LIN {X 0,Y 429.62,Z 995.465,A -85,B 0,C 180,E1 8895.717,E2 8895.717} C_VEL
LIN {X 0,Y 428.835,Z 1009.272,A -85,B 0,C 180,E1 8900.698,E2 8900.698} C_VEL
LIN {X 0,Y 428.636,Z 1016.168,A -85,B 0,C 180,E1 8904.933,E2 8904.933} C_VEL
LIN {X 0,Y 428.616,Z 1019.114,A -85,B 0,C 180,E1 8910,E2 8910} C_VEL
LIN {X 0,Y 428.715,Z 1016.175,A -85,B 0,C 180,E1 8915.065,E2 8915.065} C_VEL
LIN {X 0,Y 428.851,Z 1009.233,A -85,B 0,C 180,E1 8919.317,E2 8919.317} C_VEL
LIN {X 0,Y 429.678,Z 995.468,A -85,B 0,C 180,E1 8924.28,E2 8924.28} C_VEL
LIN {X 0,Y 431.433,Z 976.764,A -85,B 0,C 180,E1 8928.853,E2 8928.853} C_VEL
LIN {X 0,Y 434.387,Z 952.802,A -85,B 0,C 180,E1 8933.087,E2 8933.087} C_VEL
LIN {X 0,Y 438.277,Z 923.802,A -85,B 0,C 180,E1 8936.824,E2 8936.824} C_VEL
LIN {X 0,Y 442.644,Z 891.156,A -85,B 0,C 180,E1 8939.875,E2 8939.875} C_VEL
LIN {X 0,Y 446.524,Z 856.568,A -85,B 0,C 180,E1 8942.13,E2 8942.13} C_VEL
LIN {X 0,Y 449.583,Z 820.465,A -85,B 0,C 180,E1 8943.637,E2 8943.637} C_VEL
LIN {X 0,Y 450.41,Z 794.271,A -85,B 0,C 180,E1 8944.326,E2 8944.326} C_VEL
LIN {X 0,Y 439.203,Z 761.451,A -85,B 0,C 180,E1 8945.976,E2 8945.976} C_VEL
LIN {X 0,Y 430.955,Z 742.619,A -85,B 0,C 180,E1 8947.153,E2 8947.153} C_VEL
LIN {X 0,Y 427.18,Z 733.66,A -85,B 0,C 180,E1 8947.767,E2 8947.767} C_VEL
LIN {X 0,Y 427.055,Z 733.66,A -85,B 0,C 180,E1 8954.849,E2 8954.849} C_VEL
LIN {X 0,Y 427.009,Z 733.66,A -85,B 0,C 180,E1 8961.267,E2 8961.267} C_VEL
LIN {X 0,Y 427.177,Z 733.66,A -85,B 0,C 180,E1 8968.283,E2 8968.283} C_VEL
LIN {X 0,Y 427.333,Z 734.394,A -85,B 0,C 180,E1 8973.698,E2 8973.698} C_VEL
LIN {X 0,Y 436.898,Z 759.131,A -85,B 0,C 180,E1 8975.578,E2 8975.578} C_VEL
LIN {X 0,Y 439.517,Z 771.894,A -85,B 0,C 180,E1 8976.207,E2 8976.207} C_VEL
LIN {X 0,Y 438.674,Z 800.731,A -85,B 0,C 180,E1 8977.463,E2 8977.463} C_VEL
LIN {X 0,Y 437.062,Z 826.317,A -85,B 0,C 180,E1 8979.38,E2 8979.38} C_VEL
LIN {X 0,Y 435.066,Z 849.12,A -85,B 0,C 180,E1 8982.015,E2 8982.015} C_VEL
LIN {X 0,Y 433.123,Z 867.039,A -85,B 0,C 180,E1 8985.093,E2 8985.093} C_VEL
LIN {X 0,Y 431.622,Z 879.714,A -85,B 0,C 180,E1 8988.42,E2 8988.42} C_VEL
LIN {X 0,Y 430.66,Z 887.62,A -85,B 0,C 180,E1 8991.921,E2 8991.921} C_VEL
LIN {X 0,Y 430.105,Z 890.96,A -85,B 0,C 180,E1 8995.967,E2 8995.967} C_VEL
LIN {X 0,Y 430.036,Z 888.324,A -85,B 0,C 180,E1 9000.005,E2 9000.005} C_VEL
LIN {X 0,Y 430.501,Z 879.672,A -85,B 0,C 180,E1 9004.038,E2 9004.038} C_VEL
LIN {X 0,Y 431.437,Z 865.002,A -85,B 0,C 180,E1 9007.82,E2 9007.82} C_VEL
LIN {X 0,Y 432.768,Z 846,A -85,B 0,C 180,E1 9011.013,E2 9011.013} C_VEL
LIN {X 0,Y 434.452,Z 821.904,A -85,B 0,C 180,E1 9013.738,E2 9013.738} C_VEL
LIN {X 0,Y 436.003,Z 794.969,A -85,B 0,C 180,E1 9015.745,E2 9015.745} C_VEL
LIN {X 0,Y 436.384,Z 764.977,A -85,B 0,C 180,E1 9017.084,E2 9017.084} C_VEL
LIN {X 0,Y 427.56,Z 733.66,A -85,B 0,C 180,E1 9018.342,E2 9018.342} C_VEL
LIN {X 0,Y 427.307,Z 733.66,A -85,B 0,C 180,E1 9025.167,E2 9025.167} C_VEL
LIN {X 0,Y 427.11,Z 733.66,A -85,B 0,C 180,E1 9032.127,E2 9032.127} C_VEL
LIN {X 0,Y 426.99,Z 733.66,A -85,B 0,C 180,E1 9038.73,E2 9038.73} C_VEL
LIN {X 0,Y 427.072,Z 733.66,A -85,B 0,C 180,E1 9045.161,E2 9045.161} C_VEL
LIN {X 0,Y 427.062,Z 733.66,A -85,B 0,C 180,E1 9051.262,E2 9051.262} C_VEL
LIN {X 0,Y 427.143,Z 733.808,A -85,B 0,C 180,E1 9052.71,E2 9052.71} C_VEL
LIN {X 0,Y 447.309,Z 778.034,A -85,B 0,C 180,E1 9055.746,E2 9055.746} C_VEL
LIN {X 0,Y 450.534,Z 788.772,A -85,B 0,C 180,E1 9056.452,E2 9056.452} C_VEL
LIN {X 0,Y 447.329,Z 824.927,A -85,B 0,C 180,E1 9058.189,E2 9058.189} C_VEL
LIN {X 0,Y 443.379,Z 857.575,A -85,B 0,C 180,E1 9060.541,E2 9060.541} C_VEL
LIN {X 0,Y 438.938,Z 889.11,A -85,B 0,C 180,E1 9063.751,E2 9063.751} C_VEL
LIN {X 0,Y 434.909,Z 915.634,A -85,B 0,C 180,E1 9067.484,E2 9067.484} C_VEL
LIN {X 0,Y 431.753,Z 938.347,A -85,B 0,C 180,E1 9071.867,E2 9071.867} C_VEL
LIN {X 0,Y 429.91,Z 954.579,A -85,B 0,C 180,E1 9076.248,E2 9076.248} C_VEL
LIN {X 0,Y 428.868,Z 966.988,A -85,B 0,C 180,E1 9081.32,E2 9081.32} C_VEL
LIN {X 0,Y 428.48,Z 973.228,A -85,B 0,C 180,E1 9085.948,E2 9085.948} C_VEL
LIN {X 0,Y 428.501,Z 974.969,A -85,B 0,C 180,E1 9090,E2 9090} C_VEL
LIN {X 0,Y 428.596,Z 972.164,A -85,B 0,C 180,E1 9095.067,E2 9095.067} C_VEL
LIN {X 0,Y 429.066,Z 963.789,A -85,B 0,C 180,E1 9100.163,E2 9100.163} C_VEL
LIN {X 0,Y 430.461,Z 949.55,A -85,B 0,C 180,E1 9105.186,E2 9105.186} C_VEL
LIN {X 0,Y 432.926,Z 929.98,A -85,B 0,C 180,E1 9109.822,E2 9109.822} C_VEL
LIN {X 0,Y 436.34,Z 906.823,A -85,B 0,C 180,E1 9113.79,E2 9113.79} C_VEL
LIN {X 0,Y 440.492,Z 878.424,A -85,B 0,C 180,E1 9117.37,E2 9117.37} C_VEL
LIN {X 0,Y 444.819,Z 846.282,A -85,B 0,C 180,E1 9120.278,E2 9120.278} C_VEL
LIN {X 0,Y 448.724,Z 811.15,A -85,B 0,C 180,E1 9122.48,E2 9122.48} C_VEL
LIN {X 0,Y 450.013,Z 785.177,A -85,B 0,C 180,E1 9123.646,E2 9123.646} C_VEL
LIN {X 0,Y 435.647,Z 751.744,A -85,B 0,C 180,E1 9125.98,E2 9125.98} C_VEL
LIN {X 0,Y 427.221,Z 735.109,A -85,B 0,C 180,E1 9127.157,E2 9127.157} C_VEL
LIN {X 0,Y 427.068,Z 733.66,A -85,B 0,C 180,E1 9127.278,E2 9127.278} C_VEL
LIN {X 0,Y 426.949,Z 733.66,A -85,B 0,C 180,E1 9132.361,E2 9132.361} C_VEL
LIN {X 0,Y 427.02,Z 733.66,A -85,B 0,C 180,E1 9138.125,E2 9138.125} C_VEL
LIN {X 0,Y 426.978,Z 733.66,A -85,B 0,C 180,E1 9144.647,E2 9144.647} C_VEL
LIN {X 0,Y 427.157,Z 733.66,A -85,B 0,C 180,E1 9150.245,E2 9150.245} C_VEL
LIN {X 0,Y 427.426,Z 733.66,A -85,B 0,C 180,E1 9157.075,E2 9157.075} C_VEL
LIN {X 0,Y 427.537,Z 733.66,A -85,B 0,C 180,E1 9163.538,E2 9163.538} C_VEL
LIN {X 0,Y 427.72,Z 733.66,A -85,B 0,C 180,E1 9169.801,E2 9169.801} C_VEL
LIN {X 0,Y 427.981,Z 733.66,A -85,B 0,C 180,E1 9175.938,E2 9175.938} C_VEL
LIN {X 0,Y 428.158,Z 733.66,A -85,B 0,C 180,E1 9182.022,E2 9182.022} C_VEL
LIN {X 0,Y 427.902,Z 733.66,A -85,B 0,C 180,E1 9188.132,E2 9188.132} C_VEL
LIN {X 0,Y 427.634,Z 733.66,A -85,B 0,C 180,E1 9194.344,E2 9194.344} C_VEL
LIN {X 0,Y 427.461,Z 733.66,A -85,B 0,C 180,E1 9200.739,E2 9200.739} C_VEL
LIN {X 0,Y 427.215,Z 733.66,A -85,B 0,C 180,E1 9207.621,E2 9207.621} C_VEL
LIN {X 0,Y 427.13,Z 733.66,A -85,B 0,C 180,E1 9212.114,E2 9212.114} C_VEL
LIN {X 0,Y 427.002,Z 733.66,A -85,B 0,C 180,E1 9218.731,E2 9218.731} C_VEL
LIN {X 0,Y 427.058,Z 733.66,A -85,B 0,C 180,E1 9225.15,E2 9225.15} C_VEL
LIN {X 0,Y 427.107,Z 733.897,A -85,B 0,C 180,E1 9231.466,E2 9231.466} C_VEL
LIN {X 0,Y 432.238,Z 750.851,A -85,B 0,C 180,E1 9233.148,E2 9233.148} C_VEL
LIN {X 0,Y 450.687,Z 796.372,A -85,B 0,C 180,E1 9235.749,E2 9235.749} C_VEL
LIN {X 0,Y 448.347,Z 834.861,A -85,B 0,C 180,E1 9236.858,E2 9236.858} C_VEL
LIN {X 0,Y 444.853,Z 871.232,A -85,B 0,C 180,E1 9238.714,E2 9238.714} C_VEL
LIN {X 0,Y 440.772,Z 904.595,A -85,B 0,C 180,E1 9241.255,E2 9241.255} C_VEL
LIN {X 0,Y 438.262,Z 924.239,A -85,B 0,C 180,E1 9243.228,E2 9243.228} C_VEL
LIN {X 0,Y 432.759,Z 937.431,A -85,B 0,C 180,E1 9244.58,E2 9244.58} C_VEL
LIN {X 0,Y 427.29,Z 949.619,A -85,B 0,C 180,E1 9246.076,E2 9246.076} C_VEL
LIN {X 0,Y 423.868,Z 974.702,A -85,B 0,C 180,E1 9250.434,E2 9250.434} C_VEL
LIN {X 0,Y 421.981,Z 993.278,A -85,B 0,C 180,E1 9254.922,E2 9254.922} C_VEL
LIN {X 0,Y 421.01,Z 1006.872,A -85,B 0,C 180,E1 9259.641,E2 9259.641} C_VEL
LIN {X 0,Y 420.806,Z 1014.518,A -85,B 0,C 180,E1 9263.803,E2 9263.803} C_VEL
LIN {X 0,Y 420.727,Z 1018.197,A -85,B 0,C 180,E1 9267.937,E2 9267.937} C_VEL
LIN {X 0,Y 420.782,Z 1018.2,A -85,B 0,C 180,E1 9272.062,E2 9272.062} C_VEL
LIN {X 0,Y 420.831,Z 1014.521,A -85,B 0,C 180,E1 9276.196,E2 9276.196} C_VEL
LIN {X 0,Y 421.111,Z 1005.688,A -85,B 0,C 180,E1 9280.88,E2 9280.88} C_VEL
LIN {X 0,Y 422.213,Z 991.417,A -85,B 0,C 180,E1 9285.602,E2 9285.602} C_VEL
LIN {X 0,Y 424.287,Z 972.026,A -85,B 0,C 180,E1 9290.088,E2 9290.088} C_VEL
LIN {X 0,Y 427.631,Z 947.059,A -85,B 0,C 180,E1 9294.305,E2 9294.305} C_VEL
LIN {X 0,Y 431.967,Z 917.463,A -85,B 0,C 180,E1 9297.957,E2 9297.957} C_VEL
LIN {X 0,Y 436.387,Z 884.522,A -85,B 0,C 180,E1 9300.883,E2 9300.883} C_VEL
LIN {X 0,Y 440.438,Z 850.053,A -85,B 0,C 180,E1 9302.998,E2 9302.998} C_VEL
LIN {X 0,Y 443.508,Z 813.432,A -85,B 0,C 180,E1 9304.409,E2 9304.409} C_VEL
LIN {X 0,Y 443.534,Z 795.94,A -85,B 0,C 180,E1 9304.889,E2 9304.889} C_VEL
LIN {X 0,Y 428.338,Z 752.606,A -85,B 0,C 180,E1 9307.211,E2 9307.211} C_VEL
LIN {X 0,Y 419.338,Z 735.173,A -85,B 0,C 180,E1 9308.514,E2 9308.514} C_VEL
LIN {X 0,Y 419.164,Z 733.66,A -85,B 0,C 180,E1 9308.629,E2 9308.629} C_VEL
LIN {X 0,Y 419.055,Z 733.66,A -85,B 0,C 180,E1 9313.739,E2 9313.739} C_VEL
LIN {X 0,Y 419.029,Z 733.66,A -85,B 0,C 180,E1 9319.437,E2 9319.437} C_VEL
LIN {X 0,Y 419.113,Z 733.66,A -85,B 0,C 180,E1 9326.191,E2 9326.191} C_VEL
LIN {X 0,Y 419.324,Z 734.004,A -85,B 0,C 180,E1 9332.742,E2 9332.742} C_VEL
LIN {X 0,Y 429.249,Z 758.43,A -85,B 0,C 180,E1 9334.895,E2 9334.895} C_VEL
LIN {X 0,Y 432.623,Z 773.09,A -85,B 0,C 180,E1 9335.724,E2 9335.724} C_VEL
LIN {X 0,Y 431.759,Z 800.714,A -85,B 0,C 180,E1 9336.932,E2 9336.932} C_VEL
LIN {X 0,Y 429.893,Z 828.224,A -85,B 0,C 180,E1 9339.02,E2 9339.02} C_VEL
LIN {X 0,Y 427.74,Z 850.763,A -85,B 0,C 180,E1 9341.696,E2 9341.696} C_VEL
LIN {X 0,Y 425.673,Z 868.436,A -85,B 0,C 180,E1 9344.798,E2 9344.798} C_VEL
LIN {X 0,Y 423.799,Z 882.497,A -85,B 0,C 180,E1 9348.673,E2 9348.673} C_VEL
LIN {X 0,Y 422.951,Z 889.003,A -85,B 0,C 180,E1 9351.772,E2 9351.772} C_VEL
LIN {X 0,Y 422.339,Z 892.275,A -85,B 0,C 180,E1 9355.893,E2 9355.893} C_VEL
LIN {X 0,Y 422.258,Z 889.579,A -85,B 0,C 180,E1 9360.005,E2 9360.005} C_VEL
LIN {X 0,Y 422.729,Z 880.854,A -85,B 0,C 180,E1 9364.112,E2 9364.112} C_VEL
LIN {X 0,Y 423.718,Z 866.104,A -85,B 0,C 180,E1 9367.963,E2 9367.963} C_VEL
LIN {X 0,Y 425.079,Z 847.384,A -85,B 0,C 180,E1 9371.166,E2 9371.166} C_VEL
LIN {X 0,Y 426.841,Z 822.903,A -85,B 0,C 180,E1 9373.988,E2 9373.988} C_VEL
LIN {X 0,Y 428.47,Z 795.961,A -85,B 0,C 180,E1 9376.03,E2 9376.03} C_VEL
LIN {X 0,Y 428.889,Z 766.665,A -85,B 0,C 180,E1 9377.374,E2 9377.374} C_VEL
LIN {X 0,Y 419.596,Z 733.66,A -85,B 0,C 180,E1 9378.744,E2 9378.744} C_VEL
LIN {X 0,Y 419.319,Z 733.66,A -85,B 0,C 180,E1 9385.681,E2 9385.681} C_VEL
LIN {X 0,Y 419.213,Z 733.66,A -85,B 0,C 180,E1 9390.378,E2 9390.378} C_VEL
LIN {X 0,Y 419.069,Z 733.66,A -85,B 0,C 180,E1 9397.359,E2 9397.359} C_VEL
LIN {X 0,Y 419.036,Z 733.66,A -85,B 0,C 180,E1 9403.726,E2 9403.726} C_VEL
LIN {X 0,Y 419.178,Z 733.66,A -85,B 0,C 180,E1 9410.493,E2 9410.493} C_VEL
LIN {X 0,Y 419.171,Z 733.66,A -85,B 0,C 180,E1 9411.855,E2 9411.855} C_VEL
LIN {X 0,Y 423.632,Z 743.517,A -85,B 0,C 180,E1 9412.55,E2 9412.55} C_VEL
LIN {X 0,Y 440.069,Z 778.967,A -85,B 0,C 180,E1 9415.124,E2 9415.124} C_VEL
LIN {X 0,Y 443.8,Z 791.348,A -85,B 0,C 180,E1 9415.978,E2 9415.978} C_VEL
LIN {X 0,Y 440.506,Z 826.44,A -85,B 0,C 180,E1 9417.717,E2 9417.717} C_VEL
LIN {X 0,Y 436.22,Z 859.951,A -85,B 0,C 180,E1 9420.2,E2 9420.2} C_VEL
LIN {X 0,Y 431.797,Z 889.504,A -85,B 0,C 180,E1 9423.283,E2 9423.283} C_VEL
LIN {X 0,Y 427.524,Z 916.034,A -85,B 0,C 180,E1 9427.073,E2 9427.073} C_VEL
LIN {X 0,Y 424.149,Z 938.751,A -85,B 0,C 180,E1 9431.53,E2 9431.53} C_VEL
LIN {X 0,Y 422.165,Z 954.984,A -85,B 0,C 180,E1 9435.99,E2 9435.99} C_VEL
LIN {X 0,Y 421.018,Z 967.393,A -85,B 0,C 180,E1 9441.157,E2 9441.157} C_VEL
LIN {X 0,Y 420.595,Z 973.634,A -85,B 0,C 180,E1 9445.872,E2 9445.872} C_VEL
LIN {X 0,Y 420.642,Z 975.374,A -85,B 0,C 180,E1 9450,E2 9450} C_VEL
LIN {X 0,Y 420.723,Z 972.572,A -85,B 0,C 180,E1 9455.162,E2 9455.162} C_VEL
LIN {X 0,Y 421.244,Z 964.197,A -85,B 0,C 180,E1 9460.354,E2 9460.354} C_VEL
LIN {X 0,Y 422.567,Z 951.338,A -85,B 0,C 180,E1 9465.057,E2 9465.057} C_VEL
LIN {X 0,Y 425.071,Z 932.699,A -85,B 0,C 180,E1 9469.717,E2 9469.717} C_VEL
LIN {X 0,Y 428.748,Z 908.942,A -85,B 0,C 180,E1 9473.96,E2 9473.96} C_VEL
LIN {X 0,Y 433.049,Z 881.16,A -85,B 0,C 180,E1 9477.598,E2 9477.598} C_VEL
LIN {X 0,Y 437.642,Z 849.436,A -85,B 0,C 180,E1 9480.588,E2 9480.588} C_VEL
LIN {X 0,Y 441.684,Z 815.545,A -85,B 0,C 180,E1 9482.813,E2 9482.813} C_VEL
LIN {X 0,Y 443.481,Z 788.022,A -85,B 0,C 180,E1 9484.111,E2 9484.111} C_VEL
LIN {X 0,Y 428.795,Z 753.506,A -85,B 0,C 180,E1 9486.617,E2 9486.617} C_VEL
LIN {X 0,Y 419.109,Z 734.155,A -85,B 0,C 180,E1 9488.031,E2 9488.031} C_VEL
LIN {X 0,Y 418.978,Z 733.66,A -85,B 0,C 180,E1 9493.714,E2 9493.714} C_VEL
LIN {X 0,Y 419.052,Z 733.66,A -85,B 0,C 180,E1 9499.428,E2 9499.428} C_VEL
LIN {X 0,Y 419.072,Z 733.66,A -85,B 0,C 180,E1 9506.2,E2 9506.2} C_VEL
LIN {X 0,Y 419.279,Z 733.66,A -85,B 0,C 180,E1 9511.998,E2 9511.998} C_VEL
LIN {X 0,Y 419.574,Z 733.66,A -85,B 0,C 180,E1 9518.843,E2 9518.843} C_VEL
LIN {X 0,Y 419.623,Z 733.66,A -85,B 0,C 180,E1 9525.366,E2 9525.366} C_VEL
LIN {X 0,Y 419.963,Z 733.66,A -85,B 0,C 180,E1 9531.704,E2 9531.704} C_VEL
LIN {X 0,Y 420.351,Z 733.66,A -85,B 0,C 180,E1 9537.931,E2 9537.931} C_VEL
LIN {X 0,Y 420.214,Z 733.66,A -85,B 0,C 180,E1 9544.128,E2 9544.128} C_VEL
LIN {X 0,Y 419.891,Z 733.66,A -85,B 0,C 180,E1 9550.382,E2 9550.382} C_VEL
LIN {X 0,Y 419.708,Z 733.66,A -85,B 0,C 180,E1 9556.768,E2 9556.768} C_VEL
LIN {X 0,Y 419.426,Z 733.66,A -85,B 0,C 180,E1 9563.39,E2 9563.39} C_VEL
LIN {X 0,Y 419.219,Z 733.66,A -85,B 0,C 180,E1 9570.366,E2 9570.366} C_VEL
LIN {X 0,Y 419.07,Z 733.66,A -85,B 0,C 180,E1 9577.358,E2 9577.358} C_VEL
LIN {X 0,Y 419.031,Z 733.66,A -85,B 0,C 180,E1 9583.725,E2 9583.725} C_VEL
LIN {X 0,Y 419.192,Z 733.814,A -85,B 0,C 180,E1 9590.856,E2 9590.856} C_VEL
LIN {X 0,Y 423.075,Z 746.702,A -85,B 0,C 180,E1 9592.134,E2 9592.134} C_VEL
LIN {X 0,Y 444.084,Z 798.937,A -85,B 0,C 180,E1 9595.233,E2 9595.233} C_VEL
LIN {X 0,Y 441.447,Z 837.693,A -85,B 0,C 180,E1 9596.423,E2 9596.423} C_VEL
LIN {X 0,Y 437.706,Z 873.308,A -85,B 0,C 180,E1 9598.331,E2 9598.331} C_VEL
LIN {X 0,Y 433.381,Z 906.869,A -85,B 0,C 180,E1 9600.99,E2 9600.99} C_VEL
LIN {X 0,Y 428.925,Z 937.933,A -85,B 0,C 180,E1 9604.439,E2 9604.439} C_VEL
LIN {X 0,Y 427.29,Z 949.619,A -85,B 0,C 180,E1 9606.076,E2 9606.076} C_VEL
LIN {X 0,Y 421.86,Z 961.101,A -85,B 0,C 180,E1 9607.722,E2 9607.722} C_VEL
LIN {X 0,Y 416.645,Z 971.512,A -85,B 0,C 180,E1 9609.507,E2 9609.507} C_VEL
LIN {X 0,Y 414.37,Z 990.998,A -85,B 0,C 180,E1 9614.094,E2 9614.094} C_VEL
LIN {X 0,Y 413.211,Z 1005.279,A -85,B 0,C 180,E1 9618.908,E2 9618.908} C_VEL
LIN {X 0,Y 412.911,Z 1014.109,A -85,B 0,C 180,E1 9623.684,E2 9623.684} C_VEL
LIN {X 0,Y 412.83,Z 1017.79,A -85,B 0,C 180,E1 9627.898,E2 9627.898} C_VEL
LIN {X 0,Y 412.885,Z 1017.794,A -85,B 0,C 180,E1 9632.101,E2 9632.101} C_VEL
LIN {X 0,Y 413.004,Z 1012.674,A -85,B 0,C 180,E1 9637.283,E2 9637.283} C_VEL
LIN {X 0,Y 413.405,Z 1002.552,A -85,B 0,C 180,E1 9642.157,E2 9642.157} C_VEL
LIN {X 0,Y 414.797,Z 987.021,A -85,B 0,C 180,E1 9646.978,E2 9646.978} C_VEL
LIN {X 0,Y 417.523,Z 965.563,A -85,B 0,C 180,E1 9651.642,E2 9651.642} C_VEL
LIN {X 0,Y 421.355,Z 939.344,A -85,B 0,C 180,E1 9655.789,E2 9655.789} C_VEL
LIN {X 0,Y 426.153,Z 908.359,A -85,B 0,C 180,E1 9659.357,E2 9659.357} C_VEL
LIN {X 0,Y 430.704,Z 874.586,A -85,B 0,C 180,E1 9662.12,E2 9662.12} C_VEL
LIN {X 0,Y 434.776,Z 839.093,A -85,B 0,C 180,E1 9664.071,E2 9664.071} C_VEL
LIN {X 0,Y 437.646,Z 799.968,A -85,B 0,C 180,E1 9665.328,E2 9665.328} C_VEL
LIN {X 0,Y 422.889,Z 757.148,A -85,B 0,C 180,E1 9667.675,E2 9667.675} C_VEL
LIN {X 0,Y 411.388,Z 735.064,A -85,B 0,C 180,E1 9669.397,E2 9669.397} C_VEL
LIN {X 0,Y 411.261,Z 733.66,A -85,B 0,C 180,E1 9669.572,E2 9669.572} C_VEL
LIN {X 0,Y 411.079,Z 733.66,A -85,B 0,C 180,E1 9675.598,E2 9675.598} C_VEL
LIN {X 0,Y 411.059,Z 733.66,A -85,B 0,C 180,E1 9681.24,E2 9681.24} C_VEL
LIN {X 0,Y 411.205,Z 733.66,A -85,B 0,C 180,E1 9687.873,E2 9687.873} C_VEL
LIN {X 0,Y 411.363,Z 734.461,A -85,B 0,C 180,E1 9691.69,E2 9691.69} C_VEL
LIN {X 0,Y 421.291,Z 756.902,A -85,B 0,C 180,E1 9694.065,E2 9694.065} C_VEL
LIN {X 0,Y 425.852,Z 774.378,A -85,B 0,C 180,E1 9695.207,E2 9695.207} C_VEL
LIN {X 0,Y 424.792,Z 803.275,A -85,B 0,C 180,E1 9696.531,E2 9696.531} C_VEL
LIN {X 0,Y 422.819,Z 829.649,A -85,B 0,C 180,E1 9698.598,E2 9698.598} C_VEL
LIN {X 0,Y 420.454,Z 852.509,A -85,B 0,C 180,E1 9701.367,E2 9701.367} C_VEL
LIN {X 0,Y 418.285,Z 869.535,A -85,B 0,C 180,E1 9704.418,E2 9704.418} C_VEL
LIN {X 0,Y 416.438,Z 882.64,A -85,B 0,C 180,E1 9707.991,E2 9707.991} C_VEL
LIN {X 0,Y 415.263,Z 890.407,A -85,B 0,C 180,E1 9711.619,E2 9711.619} C_VEL
LIN {X 0,Y 414.583,Z 893.604,A -85,B 0,C 180,E1 9715.816,E2 9715.816} C_VEL
LIN {X 0,Y 414.474,Z 890.838,A -85,B 0,C 180,E1 9720.005,E2 9720.005} C_VEL
LIN {X 0,Y 414.956,Z 882.036,A -85,B 0,C 180,E1 9724.189,E2 9724.189} C_VEL
LIN {X 0,Y 415.973,Z 867.209,A -85,B 0,C 180,E1 9728.113,E2 9728.113} C_VEL
LIN {X 0,Y 417.424,Z 848.177,A -85,B 0,C 180,E1 9731.406,E2 9731.406} C_VEL
LIN {X 0,Y 419.248,Z 823.861,A -85,B 0,C 180,E1 9734.247,E2 9734.247} C_VEL
LIN {X 0,Y 420.929,Z 796.841,A -85,B 0,C 180,E1 9736.325,E2 9736.325} C_VEL
LIN {X 0,Y 421.325,Z 768.021,A -85,B 0,C 180,E1 9737.681,E2 9737.681} C_VEL
LIN {X 0,Y 411.642,Z 733.66,A -85,B 0,C 180,E1 9739.087,E2 9739.087} C_VEL
LIN {X 0,Y 411.343,Z 733.66,A -85,B 0,C 180,E1 9746.216,E2 9746.216} C_VEL
LIN {X 0,Y 411.195,Z 733.66,A -85,B 0,C 180,E1 9753.53,E2 9753.53} C_VEL
LIN {X 0,Y 411.043,Z 733.66,A -85,B 0,C 180,E1 9759.327,E2 9759.327} C_VEL
LIN {X 0,Y 411.107,Z 733.66,A -85,B 0,C 180,E1 9765.592,E2 9765.592} C_VEL
LIN {X 0,Y 411.259,Z 733.66,A -85,B 0,C 180,E1 9770.976,E2 9770.976} C_VEL
LIN {X 0,Y 415.774,Z 743.704,A -85,B 0,C 180,E1 9771.713,E2 9771.713} C_VEL
LIN {X 0,Y 432.504,Z 778.995,A -85,B 0,C 180,E1 9774.408,E2 9774.408} C_VEL
LIN {X 0,Y 437.157,Z 793.233,A -85,B 0,C 180,E1 9775.462,E2 9775.462} C_VEL
LIN {X 0,Y 433.608,Z 828.743,A -85,B 0,C 180,E1 9777.278,E2 9777.278} C_VEL
LIN {X 0,Y 428.927,Z 863.212,A -85,B 0,C 180,E1 9779.937,E2 9779.937} C_VEL
LIN {X 0,Y 424.097,Z 893.036,A -85,B 0,C 180,E1 9783.198,E2 9783.198} C_VEL
LIN {X 0,Y 419.752,Z 918.957,A -85,B 0,C 180,E1 9787.079,E2 9787.079} C_VEL
LIN {X 0,Y 416.22,Z 941.353,A -85,B 0,C 180,E1 9791.715,E2 9791.715} C_VEL
LIN {X 0,Y 414.179,Z 957.198,A -85,B 0,C 180,E1 9796.366,E2 9796.366} C_VEL
LIN {X 0,Y 413.096,Z 968.823,A -85,B 0,C 180,E1 9801.57,E2 9801.57} C_VEL
LIN {X 0,Y 412.712,Z 974.04,A -85,B 0,C 180,E1 9805.793,E2 9805.793} C_VEL
LIN {X 0,Y 412.751,Z 975.78,A -85,B 0,C 180,E1 9810,E2 9810} C_VEL
LIN {X 0,Y 412.836,Z 972.98,A -85,B 0,C 180,E1 9815.261,E2 9815.261} C_VEL
LIN {X 0,Y 413.404,Z 964.607,A -85,B 0,C 180,E1 9820.552,E2 9820.552} C_VEL
LIN {X 0,Y 414.864,Z 951.748,A -85,B 0,C 180,E1 9825.343,E2 9825.343} C_VEL
LIN {X 0,Y 417.571,Z 932.819,A -85,B 0,C 180,E1 9830.148,E2 9830.148} C_VEL
LIN {X 0,Y 421.453,Z 909.342,A -85,B 0,C 180,E1 9834.403,E2 9834.403} C_VEL
LIN {X 0,Y 426.023,Z 881.561,A -85,B 0,C 180,E1 9838.094,E2 9838.094} C_VEL
LIN {X 0,Y 430.87,Z 849.616,A -85,B 0,C 180,E1 9841.14,E2 9841.14} C_VEL
LIN {X 0,Y 435.13,Z 815.242,A -85,B 0,C 180,E1 9843.415,E2 9843.415} C_VEL
LIN {X 0,Y 436.69,Z 790.19,A -85,B 0,C 180,E1 9844.633,E2 9844.633} C_VEL
LIN {X 0,Y 422.715,Z 756.987,A -85,B 0,C 180,E1 9847.156,E2 9847.156} C_VEL
LIN {X 0,Y 411.359,Z 735.367,A -85,B 0,C 180,E1 9848.862,E2 9848.862} C_VEL
LIN {X 0,Y 411.165,Z 733.66,A -85,B 0,C 180,E1 9849,E2 9849} C_VEL
LIN {X 0,Y 411.042,Z 733.66,A -85,B 0,C 180,E1 9855.58,E2 9855.58} C_VEL
LIN {X 0,Y 411.074,Z 733.66,A -85,B 0,C 180,E1 9861.23,E2 9861.23} C_VEL
LIN {X 0,Y 411.171,Z 733.66,A -85,B 0,C 180,E1 9867.882,E2 9867.882} C_VEL
LIN {X 0,Y 411.395,Z 733.66,A -85,B 0,C 180,E1 9873.787,E2 9873.787} C_VEL
LIN {X 0,Y 411.703,Z 733.66,A -85,B 0,C 180,E1 9880.667,E2 9880.667} C_VEL
LIN {X 0,Y 411.732,Z 733.66,A -85,B 0,C 180,E1 9887.249,E2 9887.249} C_VEL
LIN {X 0,Y 412.16,Z 733.66,A -85,B 0,C 180,E1 9893.668,E2 9893.668} C_VEL
LIN {X 0,Y 412.456,Z 733.66,A -85,B 0,C 180,E1 9899.995,E2 9899.995} C_VEL
LIN {X 0,Y 412.113,Z 733.66,A -85,B 0,C 180,E1 9906.323,E2 9906.323} C_VEL
LIN {X 0,Y 411.87,Z 733.66,A -85,B 0,C 180,E1 9912.737,E2 9912.737} C_VEL
LIN {X 0,Y 411.664,Z 733.66,A -85,B 0,C 180,E1 9919.324,E2 9919.324} C_VEL
LIN {X 0,Y 411.374,Z 733.66,A -85,B 0,C 180,E1 9926.204,E2 9926.204} C_VEL
LIN {X 0,Y 411.199,Z 733.66,A -85,B 0,C 180,E1 9933.519,E2 9933.519} C_VEL
LIN {X 0,Y 411.049,Z 733.66,A -85,B 0,C 180,E1 9939.327,E2 9939.327} C_VEL
LIN {X 0,Y 411.093,Z 733.66,A -85,B 0,C 180,E1 9945.59,E2 9945.59} C_VEL
LIN {X 0,Y 411.285,Z 734.304,A -85,B 0,C 180,E1 9950.288,E2 9950.288} C_VEL
LIN {X 0,Y 414.481,Z 743.894,A -85,B 0,C 180,E1 9951.152,E2 9951.152} C_VEL
LIN {X 0,Y 437.548,Z 801.528,A -85,B 0,C 180,E1 9954.705,E2 9954.705} C_VEL
LIN {X 0,Y 434.621,Z 839.175,A -85,B 0,C 180,E1 9955.924,E2 9955.924} C_VEL
LIN {X 0,Y 430.641,Z 874.962,A -85,B 0,C 180,E1 9957.909,E2 9957.909} C_VEL
LIN {X 0,Y 425.975,Z 908.931,A -85,B 0,C 180,E1 9960.694,E2 9960.694} C_VEL
LIN {X 0,Y 421.318,Z 939.315,A -85,B 0,C 180,E1 9964.207,E2 9964.207} C_VEL
LIN {X 0,Y 417.525,Z 965.576,A -85,B 0,C 180,E1 9968.362,E2 9968.362} C_VEL
LIN {X 0,Y 416.645,Z 971.512,A -85,B 0,C 180,E1 9969.507,E2 9969.507} C_VEL
LIN {X 0,Y 411.549,Z 981.039,A -85,B 0,C 180,E1 9971.425,E2 9971.425} C_VEL
LIN {X 0,Y 406.706,Z 989.452,A -85,B 0,C 180,E1 9973.471,E2 9973.471} C_VEL
LIN {X 0,Y 405.366,Z 1004.869,A -85,B 0,C 180,E1 9978.691,E2 9978.691} C_VEL
LIN {X 0,Y 405.03,Z 1013.701,A -85,B 0,C 180,E1 9983.561,E2 9983.561} C_VEL
LIN {X 0,Y 404.934,Z 1017.383,A -85,B 0,C 180,E1 9987.857,E2 9987.857} C_VEL
LIN {X 0,Y 404.988,Z 1017.387,A -85,B 0,C 180,E1 9992.142,E2 9992.142} C_VEL
LIN {X 0,Y 405.119,Z 1012.479,A -85,B 0,C 180,E1 9997.282,E2 9997.282} C_VEL
LIN {X 0,Y 405.552,Z 1002.141,A -85,B 0,C 180,E1 10002.396,E2 10002.396} C_VEL
LIN {X 0,Y 407.054,Z 986.608,A -85,B 0,C 180,E1 10007.311,E2 10007.311} C_VEL
LIN {X 0,Y 409.909,Z 965.671,A -85,B 0,C 180,E1 10011.965,E2 10011.965} C_VEL
LIN {X 0,Y 413.977,Z 939.431,A -85,B 0,C 180,E1 10016.209,E2 10016.209} C_VEL
LIN {X 0,Y 418.997,Z 908.943,A -85,B 0,C 180,E1 10019.801,E2 10019.801} C_VEL
LIN {X 0,Y 423.761,Z 875.474,A -85,B 0,C 180,E1 10022.61,E2 10022.61} C_VEL
LIN {X 0,Y 428.113,Z 839.439,A -85,B 0,C 180,E1 10024.638,E2 10024.638} C_VEL
LIN {X 0,Y 430.693,Z 801.165,A -85,B 0,C 180,E1 10025.95,E2 10025.95} C_VEL
LIN {X 0,Y 417.193,Z 761.22,A -85,B 0,C 180,E1 10028.19,E2 10028.19} C_VEL
LIN {X 0,Y 403.37,Z 734.625,A -85,B 0,C 180,E1 10030.348,E2 10030.348} C_VEL
LIN {X 0,Y 403.24,Z 733.66,A -85,B 0,C 180,E1 10030.77,E2 10030.77} C_VEL
LIN {X 0,Y 403.15,Z 733.66,A -85,B 0,C 180,E1 10037.476,E2 10037.476} C_VEL
LIN {X 0,Y 403.133,Z 733.66,A -85,B 0,C 180,E1 10043.072,E2 10043.072} C_VEL
LIN {X 0,Y 403.291,Z 733.81,A -85,B 0,C 180,E1 10050.34,E2 10050.34} C_VEL
LIN {X 0,Y 413.189,Z 755.138,A -85,B 0,C 180,E1 10053.074,E2 10053.074} C_VEL
LIN {X 0,Y 419.197,Z 775.164,A -85,B 0,C 180,E1 10054.64,E2 10054.64} C_VEL
LIN {X 0,Y 417.837,Z 806.374,A -85,B 0,C 180,E1 10056.134,E2 10056.134} C_VEL
LIN {X 0,Y 415.767,Z 831.816,A -85,B 0,C 180,E1 10058.216,E2 10058.216} C_VEL
LIN {X 0,Y 413.19,Z 854.312,A -85,B 0,C 180,E1 10061.027,E2 10061.027} C_VEL
LIN {X 0,Y 410.738,Z 871.891,A -85,B 0,C 180,E1 10064.283,E2 10064.283} C_VEL
LIN {X 0,Y 408.606,Z 885.464,A -85,B 0,C 180,E1 10068.246,E2 10068.246} C_VEL
LIN {X 0,Y 407.279,Z 893.163,A -85,B 0,C 180,E1 10072.529,E2 10072.529} C_VEL
LIN {X 0,Y 406.816,Z 894.94,A -85,B 0,C 180,E1 10075.736,E2 10075.736} C_VEL
LIN {X 0,Y 406.667,Z 892.084,A -85,B 0,C 180,E1 10080.005,E2 10080.005} C_VEL
LIN {X 0,Y 407.164,Z 883.193,A -85,B 0,C 180,E1 10084.27,E2 10084.27} C_VEL
LIN {X 0,Y 408.228,Z 868.293,A -85,B 0,C 180,E1 10088.268,E2 10088.268} C_VEL
LIN {X 0,Y 409.756,Z 849.18,A -85,B 0,C 180,E1 10091.623,E2 10091.623} C_VEL
LIN {X 0,Y 411.674,Z 824.816,A -85,B 0,C 180,E1 10094.514,E2 10094.514} C_VEL
LIN {X 0,Y 413.401,Z 797.72,A -85,B 0,C 180,E1 10096.631,E2 10096.631} C_VEL
LIN {X 0,Y 413.868,Z 769.791,A -85,B 0,C 180,E1 10097.978,E2 10097.978} C_VEL
LIN {X 0,Y 403.713,Z 733.66,A -85,B 0,C 180,E1 10099.519,E2 10099.519} C_VEL
LIN {X 0,Y 403.409,Z 733.66,A -85,B 0,C 180,E1 10106.772,E2 10106.772} C_VEL
LIN {X 0,Y 403.283,Z 733.66,A -85,B 0,C 180,E1 10111.714,E2 10111.714} C_VEL
LIN {X 0,Y 403.074,Z 733.66,A -85,B 0,C 180,E1 10117.924,E2 10117.924} C_VEL
LIN {X 0,Y 403.187,Z 733.66,A -85,B 0,C 180,E1 10124.479,E2 10124.479} C_VEL
LIN {X 0,Y 403.28,Z 733.66,A -85,B 0,C 180,E1 10130.032,E2 10130.032} C_VEL
LIN {X 0,Y 408.202,Z 744.134,A -85,B 0,C 180,E1 10130.873,E2 10130.873} C_VEL
LIN {X 0,Y 425.118,Z 779.35,A -85,B 0,C 180,E1 10133.692,E2 10133.692} C_VEL
LIN {X 0,Y 430.475,Z 795.545,A -85,B 0,C 180,E1 10134.944,E2 10134.944} C_VEL
LIN {X 0,Y 426.698,Z 831.479,A -85,B 0,C 180,E1 10136.853,E2 10136.853} C_VEL
LIN {X 0,Y 421.98,Z 864.131,A -85,B 0,C 180,E1 10139.448,E2 10139.448} C_VEL
LIN {X 0,Y 417,Z 893.431,A -85,B 0,C 180,E1 10142.704,E2 10142.704} C_VEL
LIN {X 0,Y 412.189,Z 920.517,A -85,B 0,C 180,E1 10146.846,E2 10146.846} C_VEL
LIN {X 0,Y 408.59,Z 941.961,A -85,B 0,C 180,E1 10151.414,E2 10151.414} C_VEL
LIN {X 0,Y 406.358,Z 958.071,A -85,B 0,C 180,E1 10156.271,E2 10156.271} C_VEL
LIN {X 0,Y 405.239,Z 969.23,A -85,B 0,C 180,E1 10161.405,E2 10161.405} C_VEL
LIN {X 0,Y 404.831,Z 974.446,A -85,B 0,C 180,E1 10165.711,E2 10165.711} C_VEL
LIN {X 0,Y 404.86,Z 976.187,A -85,B 0,C 180,E1 10170,E2 10170} C_VEL
LIN {X 0,Y 404.966,Z 973.387,A -85,B 0,C 180,E1 10175.364,E2 10175.364} C_VEL
LIN {X 0,Y 405.502,Z 966.124,A -85,B 0,C 180,E1 10180.216,E2 10180.216} C_VEL
LIN {X 0,Y 406.924,Z 953.839,A -85,B 0,C 180,E1 10185.098,E2 10185.098} C_VEL
LIN {X 0,Y 409.688,Z 935.67,A -85,B 0,C 180,E1 10189.99,E2 10189.99} C_VEL
LIN {X 0,Y 413.553,Z 913.163,A -85,B 0,C 180,E1 10194.324,E2 10194.324} C_VEL
LIN {X 0,Y 418.491,Z 885.323,A -85,B 0,C 180,E1 10198.204,E2 10198.204} C_VEL
LIN {X 0,Y 423.434,Z 854.522,A -85,B 0,C 180,E1 10201.32,E2 10201.32} C_VEL
LIN {X 0,Y 428.025,Z 820.522,A -85,B 0,C 180,E1 10203.726,E2 10203.726} C_VEL
LIN {X 0,Y 430.06,Z 792.772,A -85,B 0,C 180,E1 10205.137,E2 10205.137} C_VEL
LIN {X 0,Y 417.171,Z 761.488,A -85,B 0,C 180,E1 10207.621,E2 10207.621} C_VEL
LIN {X 0,Y 403.214,Z 734.043,A -85,B 0,C 180,E1 10209.84,E2 10209.84} C_VEL
LIN {X 0,Y 403.138,Z 733.66,A -85,B 0,C 180,E1 10215.529,E2 10215.529} C_VEL
LIN {X 0,Y 403.097,Z 733.66,A -85,B 0,C 180,E1 10222.073,E2 10222.073} C_VEL
LIN {X 0,Y 403.279,Z 733.66,A -85,B 0,C 180,E1 10228.286,E2 10228.286} C_VEL
LIN {X 0,Y 403.512,Z 733.66,A -85,B 0,C 180,E1 10235.618,E2 10235.618} C_VEL
LIN {X 0,Y 403.777,Z 733.66,A -85,B 0,C 180,E1 10242.539,E2 10242.539} C_VEL
LIN {X 0,Y 403.907,Z 733.66,A -85,B 0,C 180,E1 10249.193,E2 10249.193} C_VEL
LIN {X 0,Y 404.258,Z 733.66,A -85,B 0,C 180,E1 10255.7,E2 10255.7} C_VEL
LIN {X 0,Y 404.462,Z 733.66,A -85,B 0,C 180,E1 10262.14,E2 10262.14} C_VEL
LIN {X 0,Y 404.133,Z 733.66,A -85,B 0,C 180,E1 10268.614,E2 10268.614} C_VEL
LIN {X 0,Y 403.851,Z 733.66,A -85,B 0,C 180,E1 10275.209,E2 10275.209} C_VEL
LIN {X 0,Y 403.617,Z 733.66,A -85,B 0,C 180,E1 10282.026,E2 10282.026} C_VEL
LIN {X 0,Y 403.336,Z 733.66,A -85,B 0,C 180,E1 10289.203,E2 10289.203} C_VEL
LIN {X 0,Y 403.233,Z 733.66,A -85,B 0,C 180,E1 10294.302,E2 10294.302} C_VEL
LIN {X 0,Y 403.117,Z 733.66,A -85,B 0,C 180,E1 10301.306,E2 10301.306} C_VEL
LIN {X 0,Y 403.192,Z 733.66,A -85,B 0,C 180,E1 10307.472,E2 10307.472} C_VEL
LIN {X 0,Y 403.338,Z 734.312,A -85,B 0,C 180,E1 10309.659,E2 10309.659} C_VEL
LIN {X 0,Y 426.799,Z 792.877,A -85,B 0,C 180,E1 10313.477,E2 10313.477} C_VEL
LIN {X 0,Y 430.873,Z 805.95,A -85,B 0,C 180,E1 10314.22,E2 10314.22} C_VEL
LIN {X 0,Y 427.686,Z 842.525,A -85,B 0,C 180,E1 10315.498,E2 10315.498} C_VEL
LIN {X 0,Y 423.469,Z 877.942,A -85,B 0,C 180,E1 10317.566,E2 10317.566} C_VEL
LIN {X 0,Y 418.354,Z 911.87,A -85,B 0,C 180,E1 10320.495,E2 10320.495} C_VEL
LIN {X 0,Y 413.757,Z 940.579,A -85,B 0,C 180,E1 10323.952,E2 10323.952} C_VEL
LIN {X 0,Y 409.701,Z 967.141,A -85,B 0,C 180,E1 10328.311,E2 10328.311} C_VEL
LIN {X 0,Y 407.005,Z 986.599,A -85,B 0,C 180,E1 10332.686,E2 10332.686} C_VEL
LIN {X 0,Y 406.706,Z 989.452,A -85,B 0,C 180,E1 10333.471,E2 10333.471} C_VEL
LIN {X 0,Y 405.076,Z 993.32,A -85,B 0,C 180,E1 10334.557,E2 10334.557} C_VEL
LIN {X 0,Y 397.721,Z 1002.34,A -85,B 0,C 180,E1 10337.601,E2 10337.601} C_VEL
LIN {X 0,Y 397.575,Z 1003.075,A -85,B 0,C 180,E1 10337.899,E2 10337.899} C_VEL
LIN {X 0,Y 397.223,Z 1011.618,A -85,B 0,C 180,E1 10342.264,E2 10342.264} C_VEL
LIN {X 0,Y 397.062,Z 1015.577,A -85,B 0,C 180,E1 10345.626,E2 10345.626} C_VEL
LIN {X 0,Y 397.071,Z 1017.49,A -85,B 0,C 180,E1 10350,E2 10350} C_VEL
LIN {X 0,Y 397.175,Z 1014.546,A -85,B 0,C 180,E1 10355.468,E2 10355.468} C_VEL
LIN {X 0,Y 397.399,Z 1006.821,A -85,B 0,C 180,E1 10360.426,E2 10360.426} C_VEL
LIN {X 0,Y 398.467,Z 993.821,A -85,B 0,C 180,E1 10365.425,E2 10365.425} C_VEL
LIN {X 0,Y 400.878,Z 974.705,A -85,B 0,C 180,E1 10370.448,E2 10370.448} C_VEL
LIN {X 0,Y 404.905,Z 949.39,A -85,B 0,C 180,E1 10375.173,E2 10375.173} C_VEL
LIN {X 0,Y 409.721,Z 921.724,A -85,B 0,C 180,E1 10378.924,E2 10378.924} C_VEL
LIN {X 0,Y 415.013,Z 889.596,A -85,B 0,C 180,E1 10382.092,E2 10382.092} C_VEL
LIN {X 0,Y 419.821,Z 855.25,A -85,B 0,C 180,E1 10384.439,E2 10384.439} C_VEL
LIN {X 0,Y 423.484,Z 819.925,A -85,B 0,C 180,E1 10385.989,E2 10385.989} C_VEL
LIN {X 0,Y 423.981,Z 803.038,A -85,B 0,C 180,E1 10386.544,E2 10386.544} C_VEL
LIN {X 0,Y 411.887,Z 765.971,A -85,B 0,C 180,E1 10388.665,E2 10388.665} C_VEL
LIN {X 0,Y 398.826,Z 740.224,A -85,B 0,C 180,E1 10390.942,E2 10390.942} C_VEL
LIN {X 0,Y 395.416,Z 735.171,A -85,B 0,C 180,E1 10391.998,E2 10391.998} C_VEL
LIN {X 0,Y 395.276,Z 733.66,A -85,B 0,C 180,E1 10392.296,E2 10392.296} C_VEL
LIN {X 0,Y 395.197,Z 733.66,A -85,B 0,C 180,E1 10399.369,E2 10399.369} C_VEL
LIN {X 0,Y 395.241,Z 733.66,A -85,B 0,C 180,E1 10404.935,E2 10404.935} C_VEL
LIN {X 0,Y 395.388,Z 734.194,A -85,B 0,C 180,E1 10408.772,E2 10408.772} C_VEL
LIN {X 0,Y 404.389,Z 752.237,A -85,B 0,C 180,E1 10411.744,E2 10411.744} C_VEL
LIN {X 0,Y 411.177,Z 770.552,A -85,B 0,C 180,E1 10413.615,E2 10413.615} C_VEL
LIN {X 0,Y 412.526,Z 779.965,A -85,B 0,C 180,E1 10414.2,E2 10414.2} C_VEL
LIN {X 0,Y 411,Z 809.315,A -85,B 0,C 180,E1 10415.711,E2 10415.711} C_VEL
LIN {X 0,Y 408.637,Z 835.261,A -85,B 0,C 180,E1 10417.945,E2 10417.945} C_VEL
LIN {X 0,Y 405.713,Z 857.996,A -85,B 0,C 180,E1 10420.947,E2 10420.947} C_VEL
LIN {X 0,Y 403.049,Z 875.057,A -85,B 0,C 180,E1 10424.346,E2 10424.346} C_VEL
LIN {X 0,Y 401.033,Z 886.997,A -85,B 0,C 180,E1 10428.021,E2 10428.021} C_VEL
LIN {X 0,Y 399.865,Z 893.288,A -85,B 0,C 180,E1 10431.294,E2 10431.294} C_VEL
LIN {X 0,Y 399.061,Z 896.286,A -85,B 0,C 180,E1 10435.653,E2 10435.653} C_VEL
LIN {X 0,Y 398.884,Z 893.337,A -85,B 0,C 180,E1 10440.005,E2 10440.005} C_VEL
LIN {X 0,Y 399.393,Z 884.333,A -85,B 0,C 180,E1 10444.353,E2 10444.353} C_VEL
LIN {X 0,Y 400.499,Z 869.326,A -85,B 0,C 180,E1 10448.428,E2 10448.428} C_VEL
LIN {X 0,Y 402.135,Z 849.498,A -85,B 0,C 180,E1 10451.931,E2 10451.931} C_VEL
LIN {X 0,Y 404.078,Z 825.61,A -85,B 0,C 180,E1 10454.793,E2 10454.793} C_VEL
LIN {X 0,Y 405.958,Z 797.299,A -85,B 0,C 180,E1 10457.014,E2 10457.014} C_VEL
LIN {X 0,Y 406.293,Z 770.922,A -85,B 0,C 180,E1 10458.306,E2 10458.306} C_VEL
LIN {X 0,Y 395.764,Z 733.66,A -85,B 0,C 180,E1 10459.962,E2 10459.962} C_VEL
LIN {X 0,Y 395.422,Z 733.66,A -85,B 0,C 180,E1 10467.358,E2 10467.358} C_VEL
LIN {X 0,Y 395.299,Z 733.66,A -85,B 0,C 180,E1 10472.579,E2 10472.579} C_VEL
LIN {X 0,Y 395.204,Z 733.66,A -85,B 0,C 180,E1 10479.984,E2 10479.984} C_VEL
LIN {X 0,Y 395.266,Z 733.66,A -85,B 0,C 180,E1 10486.707,E2 10486.707} C_VEL
LIN {X 0,Y 395.332,Z 734.017,A -85,B 0,C 180,E1 10489.087,E2 10489.087} C_VEL
LIN {X 0,Y 400.454,Z 744.287,A -85,B 0,C 180,E1 10489.962,E2 10489.962} C_VEL
LIN {X 0,Y 417.599,Z 779.285,A -85,B 0,C 180,E1 10492.91,E2 10492.91} C_VEL
LIN {X 0,Y 423.821,Z 798.451,A -85,B 0,C 180,E1 10494.438,E2 10494.438} C_VEL
LIN {X 0,Y 419.821,Z 833.935,A -85,B 0,C 180,E1 10496.407,E2 10496.407} C_VEL
LIN {X 0,Y 414.856,Z 866.329,A -85,B 0,C 180,E1 10499.069,E2 10499.069} C_VEL
LIN {X 0,Y 409.658,Z 895.285,A -85,B 0,C 180,E1 10502.386,E2 10502.386} C_VEL
LIN {X 0,Y 404.645,Z 921.966,A -85,B 0,C 180,E1 10506.595,E2 10506.595} C_VEL
LIN {X 0,Y 401.01,Z 942.381,A -85,B 0,C 180,E1 10511.054,E2 10511.054} C_VEL
LIN {X 0,Y 398.585,Z 958.806,A -85,B 0,C 180,E1 10516.122,E2 10516.122} C_VEL
LIN {X 0,Y 397.408,Z 969.636,A -85,B 0,C 180,E1 10521.234,E2 10521.234} C_VEL
LIN {X 0,Y 396.949,Z 974.853,A -85,B 0,C 180,E1 10525.625,E2 10525.625} C_VEL
LIN {X 0,Y 396.969,Z 976.593,A -85,B 0,C 180,E1 10530,E2 10530} C_VEL
LIN {X 0,Y 397.092,Z 973.795,A -85,B 0,C 180,E1 10535.47,E2 10535.47} C_VEL
LIN {X 0,Y 397.763,Z 965.427,A -85,B 0,C 180,E1 10540.972,E2 10540.972} C_VEL
LIN {X 0,Y 399.474,Z 952.569,A -85,B 0,C 180,E1 10545.95,E2 10545.95} C_VEL
LIN {X 0,Y 402.591,Z 933.633,A -85,B 0,C 180,E1 10550.934,E2 10550.934} C_VEL
LIN {X 0,Y 406.956,Z 910.155,A -85,B 0,C 180,E1 10555.332,E2 10555.332} C_VEL
LIN {X 0,Y 412.034,Z 882.364,A -85,B 0,C 180,E1 10559.137,E2 10559.137} C_VEL
LIN {X 0,Y 417.464,Z 849.506,A -85,B 0,C 180,E1 10562.342,E2 10562.342} C_VEL
LIN {X 0,Y 422.108,Z 815.044,A -85,B 0,C 180,E1 10564.652,E2 10564.652} C_VEL
LIN {X 0,Y 423.344,Z 794.904,A -85,B 0,C 180,E1 10565.691,E2 10565.691} C_VEL
LIN {X 0,Y 410.532,Z 763.656,A -85,B 0,C 180,E1 10568.287,E2 10568.287} C_VEL
LIN {X 0,Y 395.278,Z 734.741,A -85,B 0,C 180,E1 10570.799,E2 10570.799} C_VEL
LIN {X 0,Y 395.19,Z 733.66,A -85,B 0,C 180,E1 10570.994,E2 10570.994} C_VEL
LIN {X 0,Y 395.192,Z 733.66,A -85,B 0,C 180,E1 10576.715,E2 10576.715} C_VEL
LIN {X 0,Y 395.187,Z 733.66,A -85,B 0,C 180,E1 10583.57,E2 10583.57} C_VEL
LIN {X 0,Y 395.408,Z 733.66,A -85,B 0,C 180,E1 10590.142,E2 10590.142} C_VEL
LIN {X 0,Y 395.675,Z 733.66,A -85,B 0,C 180,E1 10597.497,E2 10597.497} C_VEL
LIN {X 0,Y 395.827,Z 733.66,A -85,B 0,C 180,E1 10604.465,E2 10604.465} C_VEL
LIN {X 0,Y 396.162,Z 733.66,A -85,B 0,C 180,E1 10611.531,E2 10611.531} C_VEL
LIN {X 0,Y 396.625,Z 733.66,A -85,B 0,C 180,E1 10617.807,E2 10617.807} C_VEL
LIN {X 0,Y 396.454,Z 733.66,A -85,B 0,C 180,E1 10624.375,E2 10624.375} C_VEL
LIN {X 0,Y 396.117,Z 733.66,A -85,B 0,C 180,E1 10631.012,E2 10631.012} C_VEL
LIN {X 0,Y 395.88,Z 733.66,A -85,B 0,C 180,E1 10637.81,E2 10637.81} C_VEL
LIN {X 0,Y 395.544,Z 733.66,A -85,B 0,C 180,E1 10644.895,E2 10644.895} C_VEL
LIN {X 0,Y 395.407,Z 733.66,A -85,B 0,C 180,E1 10649.847,E2 10649.847} C_VEL
LIN {X 0,Y 395.186,Z 733.66,A -85,B 0,C 180,E1 10656.43,E2 10656.43} C_VEL
LIN {X 0,Y 395.223,Z 733.66,A -85,B 0,C 180,E1 10663.587,E2 10663.587} C_VEL
LIN {X 0,Y 395.308,Z 733.686,A -85,B 0,C 180,E1 10668.658,E2 10668.658} C_VEL
LIN {X 0,Y 397.681,Z 739.237,A -85,B 0,C 180,E1 10669.085,E2 10669.085} C_VEL
LIN {X 0,Y 418.062,Z 788.562,A -85,B 0,C 180,E1 10672.491,E2 10672.491} C_VEL
LIN {X 0,Y 424.308,Z 807.984,A -85,B 0,C 180,E1 10673.655,E2 10673.655} C_VEL
LIN {X 0,Y 420.764,Z 845.838,A -85,B 0,C 180,E1 10675.055,E2 10675.055} C_VEL
LIN {X 0,Y 416.235,Z 881.064,A -85,B 0,C 180,E1 10677.242,E2 10677.242} C_VEL
LIN {X 0,Y 410.997,Z 913.46,A -85,B 0,C 180,E1 10680.151,E2 10680.151} C_VEL
LIN {X 0,Y 406.146,Z 942.111,A -85,B 0,C 180,E1 10683.724,E2 10683.724} C_VEL
LIN {X 0,Y 401.919,Z 968.079,A -85,B 0,C 180,E1 10688.16,E2 10688.16} C_VEL
LIN {X 0,Y 399.039,Z 988.177,A -85,B 0,C 180,E1 10692.898,E2 10692.898} C_VEL
LIN {X 0,Y 397.575,Z 1003.075,A -85,B 0,C 180,E1 10697.899,E2 10697.899} C_VEL
LIN {X 0,Y 394.837,Z 1007.043,A -85,B 0,C 180,E1 10699.667,E2 10699.667} C_VEL
LIN {X 0,Y 389.373,Z 1011.604,A -85,B 0,C 180,E1 10702.382,E2 10702.382} C_VEL
LIN {X 0,Y 389.267,Z 1012.041,A -85,B 0,C 180,E1 10702.699,E2 10702.699} C_VEL
LIN {X 0,Y 389.162,Z 1016.57,A -85,B 0,C 180,E1 10707.77,E2 10707.77} C_VEL
LIN {X 0,Y 389.214,Z 1016.574,A -85,B 0,C 180,E1 10712.229,E2 10712.229} C_VEL
LIN {X 0,Y 389.277,Z 1012.889,A -85,B 0,C 180,E1 10716.7,E2 10716.7} C_VEL
LIN {X 0,Y 389.671,Z 1004.046,A -85,B 0,C 180,E1 10721.77,E2 10721.77} C_VEL
LIN {X 0,Y 391.114,Z 989.766,A -85,B 0,C 180,E1 10726.878,E2 10726.878} C_VEL
LIN {X 0,Y 393.939,Z 970.382,A -85,B 0,C 180,E1 10731.711,E2 10731.711} C_VEL
LIN {X 0,Y 398.219,Z 945.582,A -85,B 0,C 180,E1 10736.205,E2 10736.205} C_VEL
LIN {X 0,Y 403.714,Z 915.507,A -85,B 0,C 180,E1 10740.15,E2 10740.15} C_VEL
LIN {X 0,Y 409.165,Z 882.461,A -85,B 0,C 180,E1 10743.238,E2 10743.238} C_VEL
LIN {X 0,Y 414.331,Z 845.973,A -85,B 0,C 180,E1 10745.546,E2 10745.546} C_VEL
LIN {X 0,Y 417.995,Z 808.864,A -85,B 0,C 180,E1 10746.951,E2 10746.951} C_VEL
LIN {X 0,Y 406.766,Z 770.999,A -85,B 0,C 180,E1 10749.128,E2 10749.128} C_VEL
LIN {X 0,Y 395.612,Z 748.744,A -85,B 0,C 180,E1 10751.143,E2 10751.143} C_VEL
LIN {X 0,Y 390.424,Z 739.913,A -85,B 0,C 180,E1 10752.961,E2 10752.961} C_VEL
LIN {X 0,Y 387.334,Z 734.574,A -85,B 0,C 180,E1 10754.369,E2 10754.369} C_VEL
LIN {X 0,Y 387.221,Z 733.66,A -85,B 0,C 180,E1 10755.275,E2 10755.275} C_VEL
LIN {X 0,Y 387.263,Z 733.66,A -85,B 0,C 180,E1 10761.439,E2 10761.439} C_VEL
LIN {X 0,Y 387.325,Z 734.24,A -85,B 0,C 180,E1 10766.538,E2 10766.538} C_VEL
LIN {X 0,Y 394.207,Z 746.547,A -85,B 0,C 180,E1 10769.57,E2 10769.57} C_VEL
LIN {X 0,Y 402.23,Z 764.646,A -85,B 0,C 180,E1 10772.188,E2 10772.188} C_VEL
LIN {X 0,Y 406.216,Z 779.719,A -85,B 0,C 180,E1 10773.516,E2 10773.516} C_VEL
LIN {X 0,Y 404.388,Z 810.307,A -85,B 0,C 180,E1 10775.115,E2 10775.115} C_VEL
LIN {X 0,Y 401.756,Z 836.661,A -85,B 0,C 180,E1 10777.432,E2 10777.432} C_VEL
LIN {X 0,Y 398.793,Z 858.244,A -85,B 0,C 180,E1 10780.315,E2 10780.315} C_VEL
LIN {X 0,Y 396.064,Z 874.581,A -85,B 0,C 180,E1 10783.498,E2 10783.498} C_VEL
LIN {X 0,Y 393.783,Z 887.176,A -85,B 0,C 180,E1 10787.233,E2 10787.233} C_VEL
LIN {X 0,Y 392.169,Z 894.76,A -85,B 0,C 180,E1 10791.122,E2 10791.122} C_VEL
LIN {X 0,Y 391.292,Z 897.643,A -85,B 0,C 180,E1 10795.567,E2 10795.567} C_VEL
LIN {X 0,Y 391.098,Z 894.573,A -85,B 0,C 180,E1 10800.005,E2 10800.005} C_VEL
LIN {X 0,Y 391.512,Z 886.946,A -85,B 0,C 180,E1 10803.885,E2 10803.885} C_VEL
LIN {X 0,Y 392.443,Z 873.983,A -85,B 0,C 180,E1 10807.765,E2 10807.765} C_VEL
LIN {X 0,Y 394.103,Z 854.814,A -85,B 0,C 180,E1 10811.49,E2 10811.49} C_VEL
LIN {X 0,Y 396.065,Z 831.71,A -85,B 0,C 180,E1 10814.533,E2 10814.533} C_VEL
LIN {X 0,Y 397.992,Z 805.161,A -85,B 0,C 180,E1 10816.867,E2 10816.867} C_VEL
LIN {X 0,Y 399.334,Z 775.838,A -85,B 0,C 180,E1 10818.463,E2 10818.463} C_VEL
LIN {X 0,Y 387.795,Z 733.66,A -85,B 0,C 180,E1 10820.439,E2 10820.439} C_VEL
LIN {X 0,Y 387.516,Z 733.66,A -85,B 0,C 180,E1 10827.964,E2 10827.964} C_VEL
LIN {X 0,Y 387.315,Z 733.66,A -85,B 0,C 180,E1 10834.822,E2 10834.822} C_VEL
LIN {X 0,Y 387.198,Z 733.66,A -85,B 0,C 180,E1 10842.015,E2 10842.015} C_VEL
LIN {X 0,Y 387.35,Z 733.815,A -85,B 0,C 180,E1 10848.043,E2 10848.043} C_VEL
LIN {X 0,Y 389.801,Z 739.334,A -85,B 0,C 180,E1 10848.503,E2 10848.503} C_VEL
LIN {X 0,Y 408.407,Z 775.486,A -85,B 0,C 180,E1 10851.769,E2 10851.769} C_VEL
LIN {X 0,Y 417.342,Z 799.69,A -85,B 0,C 180,E1 10853.845,E2 10853.845} C_VEL
LIN {X 0,Y 413.29,Z 834.06,A -85,B 0,C 180,E1 10855.782,E2 10855.782} C_VEL
LIN {X 0,Y 408.077,Z 866.553,A -85,B 0,C 180,E1 10858.478,E2 10858.478} C_VEL
LIN {X 0,Y 402.54,Z 896.079,A -85,B 0,C 180,E1 10861.914,E2 10861.914} C_VEL
LIN {X 0,Y 397.273,Z 922.528,A -85,B 0,C 180,E1 10866.167,E2 10866.167} C_VEL
LIN {X 0,Y 393.327,Z 943.418,A -85,B 0,C 180,E1 10870.844,E2 10870.844} C_VEL
LIN {X 0,Y 390.761,Z 959.722,A -85,B 0,C 180,E1 10876.034,E2 10876.034} C_VEL
LIN {X 0,Y 389.557,Z 970.043,A -85,B 0,C 180,E1 10881.056,E2 10881.056} C_VEL
LIN {X 0,Y 389.082,Z 975.259,A -85,B 0,C 180,E1 10885.537,E2 10885.537} C_VEL
LIN {X 0,Y 389.089,Z 976.999,A -85,B 0,C 180,E1 10890,E2 10890} C_VEL
LIN {X 0,Y 389.206,Z 974.203,A -85,B 0,C 180,E1 10895.581,E2 10895.581} C_VEL
LIN {X 0,Y 389.967,Z 965.836,A -85,B 0,C 180,E1 10901.194,E2 10901.194} C_VEL
LIN {X 0,Y 391.788,Z 952.98,A -85,B 0,C 180,E1 10906.271,E2 10906.271} C_VEL
LIN {X 0,Y 395.126,Z 934.043,A -85,B 0,C 180,E1 10911.348,E2 10911.348} C_VEL
LIN {X 0,Y 399.742,Z 910.563,A -85,B 0,C 180,E1 10915.823,E2 10915.823} C_VEL
LIN {X 0,Y 405.095,Z 882.766,A -85,B 0,C 180,E1 10919.686,E2 10919.686} C_VEL
LIN {X 0,Y 410.771,Z 849.907,A -85,B 0,C 180,E1 10922.934,E2 10922.934} C_VEL
LIN {X 0,Y 415.546,Z 816.173,A -85,B 0,C 180,E1 10925.229,E2 10925.229} C_VEL
LIN {X 0,Y 416.805,Z 797.504,A -85,B 0,C 180,E1 10926.225,E2 10926.225} C_VEL
LIN {X 0,Y 404.356,Z 766.637,A -85,B 0,C 180,E1 10928.905,E2 10928.905} C_VEL
LIN {X 0,Y 387.351,Z 734.997,A -85,B 0,C 180,E1 10931.822,E2 10931.822} C_VEL
LIN {X 0,Y 387.226,Z 733.66,A -85,B 0,C 180,E1 10932.015,E2 10932.015} C_VEL
LIN {X 0,Y 387.206,Z 733.66,A -85,B 0,C 180,E1 10938.333,E2 10938.333} C_VEL
LIN {X 0,Y 387.321,Z 733.66,A -85,B 0,C 180,E1 10945.178,E2 10945.178} C_VEL
LIN {X 0,Y 387.542,Z 733.66,A -85,B 0,C 180,E1 10952.038,E2 10952.038} C_VEL
LIN {X 0,Y 387.862,Z 733.66,A -85,B 0,C 180,E1 10959.536,E2 10959.536} C_VEL
LIN {X 0,Y 387.945,Z 733.66,A -85,B 0,C 180,E1 10966.453,E2 10966.453} C_VEL
LIN {X 0,Y 388.431,Z 733.66,A -85,B 0,C 180,E1 10973.28,E2 10973.28} C_VEL
LIN {X 0,Y 388.759,Z 733.66,A -85,B 0,C 180,E1 10979.995,E2 10979.995} C_VEL
LIN {X 0,Y 388.403,Z 733.66,A -85,B 0,C 180,E1 10986.711,E2 10986.711} C_VEL
LIN {X 0,Y 388.066,Z 733.66,A -85,B 0,C 180,E1 10993.533,E2 10993.533} C_VEL
LIN {X 0,Y 387.813,Z 733.66,A -85,B 0,C 180,E1 11000.565,E2 11000.565} C_VEL
LIN {X 0,Y 387.53,Z 733.66,A -85,B 0,C 180,E1 11007.952,E2 11007.952} C_VEL
LIN {X 0,Y 387.327,Z 733.66,A -85,B 0,C 180,E1 11014.824,E2 11014.824} C_VEL
LIN {X 0,Y 387.203,Z 733.66,A -85,B 0,C 180,E1 11022.015,E2 11022.015} C_VEL
LIN {X 0,Y 387.409,Z 734.127,A -85,B 0,C 180,E1 11027.642,E2 11027.642} C_VEL
LIN {X 0,Y 392.911,Z 744.79,A -85,B 0,C 180,E1 11028.616,E2 11028.616} C_VEL
LIN {X 0,Y 413.023,Z 794.569,A -85,B 0,C 180,E1 11032.109,E2 11032.109} C_VEL
LIN {X 0,Y 417.838,Z 809.58,A -85,B 0,C 180,E1 11033.064,E2 11033.064} C_VEL
LIN {X 0,Y 414.046,Z 847.191,A -85,B 0,C 180,E1 11034.512,E2 11034.512} C_VEL
LIN {X 0,Y 409.231,Z 882.381,A -85,B 0,C 180,E1 11036.767,E2 11036.767} C_VEL
LIN {X 0,Y 403.852,Z 913.968,A -85,B 0,C 180,E1 11039.68,E2 11039.68} C_VEL
LIN {X 0,Y 398.49,Z 943.853,A -85,B 0,C 180,E1 11043.524,E2 11043.524} C_VEL
LIN {X 0,Y 394.159,Z 969.015,A -85,B 0,C 180,E1 11048.004,E2 11048.004} C_VEL
LIN {X 0,Y 391.064,Z 989.753,A -85,B 0,C 180,E1 11053.119,E2 11053.119} C_VEL
LIN {X 0,Y 389.626,Z 1004.043,A -85,B 0,C 180,E1 11058.228,E2 11058.228} C_VEL
LIN {X 0,Y 389.267,Z 1012.041,A -85,B 0,C 180,E1 11062.699,E2 11062.699} C_VEL
LIN {X 0,Y 386.746,Z 1014.289,A -85,B 0,C 180,E1 11064.57,E2 11064.57} C_VEL
LIN {X 0,Y 381.262,Z 1016.168,A -85,B 0,C 180,E1 11067.748,E2 11067.748} C_VEL
LIN {X 0,Y 381.318,Z 1016.167,A -85,B 0,C 180,E1 11072.275,E2 11072.275} C_VEL
LIN {X 0,Y 381.379,Z 1012.17,A -85,B 0,C 180,E1 11077.084,E2 11077.084} C_VEL
LIN {X 0,Y 381.928,Z 1002.28,A -85,B 0,C 180,E1 11082.594,E2 11082.594} C_VEL
LIN {X 0,Y 383.58,Z 987.359,A -85,B 0,C 180,E1 11087.813,E2 11087.813} C_VEL
LIN {X 0,Y 387.104,Z 965.915,A -85,B 0,C 180,E1 11093.025,E2 11093.025} C_VEL
LIN {X 0,Y 392.068,Z 939.388,A -85,B 0,C 180,E1 11097.607,E2 11097.607} C_VEL
LIN {X 0,Y 397.825,Z 909.52,A -85,B 0,C 180,E1 11101.342,E2 11101.342} C_VEL
LIN {X 0,Y 403.59,Z 875.166,A -85,B 0,C 180,E1 11104.39,E2 11104.39} C_VEL
LIN {X 0,Y 408.478,Z 840.131,A -85,B 0,C 180,E1 11106.459,E2 11106.459} C_VEL
LIN {X 0,Y 411.221,Z 808.276,A -85,B 0,C 180,E1 11107.673,E2 11107.673} C_VEL
LIN {X 0,Y 400.614,Z 773.898,A -85,B 0,C 180,E1 11109.776,E2 11109.776} C_VEL
LIN {X 0,Y 392.293,Z 756.787,A -85,B 0,C 180,E1 11111.372,E2 11111.372} C_VEL
LIN {X 0,Y 389.022,Z 749.911,A -85,B 0,C 180,E1 11112.601,E2 11112.601} C_VEL
LIN {X 0,Y 383.483,Z 740.591,A -85,B 0,C 180,E1 11115.203,E2 11115.203} C_VEL
LIN {X 0,Y 379.282,Z 734.66,A -85,B 0,C 180,E1 11119.164,E2 11119.164} C_VEL
LIN {X 0,Y 379.344,Z 733.924,A -85,B 0,C 180,E1 11121.603,E2 11121.603} C_VEL
LIN {X 0,Y 381.933,Z 739.417,A -85,B 0,C 180,E1 11125.149,E2 11125.149} C_VEL
LIN {X 0,Y 383.848,Z 741.558,A -85,B 0,C 180,E1 11126.271,E2 11126.271} C_VEL
LIN {X 0,Y 389.907,Z 752.745,A -85,B 0,C 180,E1 11129.195,E2 11129.195} C_VEL
LIN {X 0,Y 396.991,Z 769.745,A -85,B 0,C 180,E1 11131.758,E2 11131.758} C_VEL
LIN {X 0,Y 399.892,Z 782.406,A -85,B 0,C 180,E1 11132.908,E2 11132.908} C_VEL
LIN {X 0,Y 397.677,Z 813.851,A -85,B 0,C 180,E1 11134.666,E2 11134.666} C_VEL
LIN {X 0,Y 394.689,Z 840.203,A -85,B 0,C 180,E1 11137.122,E2 11137.122} C_VEL
LIN {X 0,Y 391.327,Z 862.053,A -85,B 0,C 180,E1 11140.218,E2 11140.218} C_VEL
LIN {X 0,Y 388.209,Z 878.785,A -85,B 0,C 180,E1 11143.782,E2 11143.782} C_VEL
LIN {X 0,Y 385.907,Z 890.196,A -85,B 0,C 180,E1 11147.544,E2 11147.544} C_VEL
LIN {X 0,Y 384.498,Z 896.26,A -85,B 0,C 180,E1 11150.943,E2 11150.943} C_VEL
LIN {X 0,Y 383.539,Z 899.004,A -85,B 0,C 180,E1 11155.477,E2 11155.477} C_VEL
LIN {X 0,Y 383.289,Z 895.816,A -85,B 0,C 180,E1 11160.005,E2 11160.005} C_VEL
LIN {X 0,Y 383.71,Z 888.067,A -85,B 0,C 180,E1 11163.965,E2 11163.965} C_VEL
LIN {X 0,Y 384.7,Z 874.983,A -85,B 0,C 180,E1 11167.922,E2 11167.922} C_VEL
LIN {X 0,Y 386.36,Z 856.662,A -85,B 0,C 180,E1 11171.562,E2 11171.562} C_VEL
LIN {X 0,Y 388.392,Z 833.708,A -85,B 0,C 180,E1 11174.683,E2 11174.683} C_VEL
LIN {X 0,Y 390.383,Z 807.744,A -85,B 0,C 180,E1 11177.06,E2 11177.06} C_VEL
LIN {X 0,Y 391.843,Z 777.018,A -85,B 0,C 180,E1 11178.796,E2 11178.796} C_VEL
LIN {X 0,Y 379.845,Z 733.66,A -85,B 0,C 180,E1 11180.815,E2 11180.815} C_VEL
LIN {X 0,Y 379.531,Z 733.66,A -85,B 0,C 180,E1 11188.639,E2 11188.639} C_VEL
LIN {X 0,Y 379.381,Z 733.66,A -85,B 0,C 180,E1 11193.972,E2 11193.972} C_VEL
LIN {X 0,Y 379.205,Z 733.66,A -85,B 0,C 180,E1 11200.657,E2 11200.657} C_VEL
LIN {X 0,Y 379.291,Z 733.791,A -85,B 0,C 180,E1 11206.93,E2 11206.93} C_VEL
LIN {X 0,Y 381.829,Z 739.376,A -85,B 0,C 180,E1 11207.429,E2 11207.429} C_VEL
LIN {X 0,Y 400.45,Z 774.587,A -85,B 0,C 180,E1 11210.818,E2 11210.818} C_VEL
LIN {X 0,Y 410.761,Z 802.328,A -85,B 0,C 180,E1 11213.3,E2 11213.3} C_VEL
LIN {X 0,Y 406.296,Z 837.184,A -85,B 0,C 180,E1 11215.35,E2 11215.35} C_VEL
LIN {X 0,Y 400.747,Z 870.16,A -85,B 0,C 180,E1 11218.212,E2 11218.212} C_VEL
LIN {X 0,Y 394.718,Z 900.383,A -85,B 0,C 180,E1 11221.92,E2 11221.92} C_VEL
LIN {X 0,Y 389.406,Z 925.544,A -85,B 0,C 180,E1 11226.216,E2 11226.216} C_VEL
LIN {X 0,Y 385.37,Z 945.882,A -85,B 0,C 180,E1 11231.015,E2 11231.015} C_VEL
LIN {X 0,Y 382.843,Z 961.469,A -85,B 0,C 180,E1 11236.274,E2 11236.274} C_VEL
LIN {X 0,Y 381.724,Z 970.45,A -85,B 0,C 180,E1 11240.871,E2 11240.871} C_VEL
LIN {X 0,Y 381.199,Z 975.665,A -85,B 0,C 180,E1 11245.444,E2 11245.444} C_VEL
LIN {X 0,Y 381.198,Z 977.406,A -85,B 0,C 180,E1 11250,E2 11250} C_VEL
LIN {X 0,Y 381.35,Z 974.61,A -85,B 0,C 180,E1 11255.697,E2 11255.697} C_VEL
LIN {X 0,Y 382.153,Z 966.247,A -85,B 0,C 180,E1 11261.426,E2 11261.426} C_VEL
LIN {X 0,Y 384.097,Z 953.392,A -85,B 0,C 180,E1 11266.607,E2 11266.607} C_VEL
LIN {X 0,Y 387.694,Z 934.452,A -85,B 0,C 180,E1 11271.778,E2 11271.778} C_VEL
LIN {X 0,Y 392.531,Z 910.971,A -85,B 0,C 180,E1 11276.333,E2 11276.333} C_VEL
LIN {X 0,Y 398.317,Z 882.557,A -85,B 0,C 180,E1 11280.329,E2 11280.329} C_VEL
LIN {X 0,Y 404.128,Z 850.294,A -85,B 0,C 180,E1 11283.547,E2 11283.547} C_VEL
LIN {X 0,Y 409.192,Z 816.003,A -85,B 0,C 180,E1 11285.898,E2 11285.898} C_VEL
LIN {X 0,Y 410.68,Z 801.379,A -85,B 0,C 180,E1 11286.667,E2 11286.667} C_VEL
LIN {X 0,Y 398.187,Z 769.702,A -85,B 0,C 180,E1 11289.536,E2 11289.536} C_VEL
LIN {X 0,Y 379.328,Z 734.907,A -85,B 0,C 180,E1 11292.928,E2 11292.928} C_VEL
LIN {X 0,Y 379.202,Z 733.66,A -85,B 0,C 180,E1 11293.17,E2 11293.17} C_VEL
LIN {X 0,Y 379.223,Z 733.66,A -85,B 0,C 180,E1 11300.292,E2 11300.292} C_VEL
LIN {X 0,Y 379.442,Z 733.66,A -85,B 0,C 180,E1 11306.927,E2 11306.927} C_VEL
LIN {X 0,Y 379.667,Z 733.66,A -85,B 0,C 180,E1 11313.977,E2 11313.977} C_VEL
LIN {X 0,Y 379.959,Z 733.66,A -85,B 0,C 180,E1 11321.406,E2 11321.406} C_VEL
LIN {X 0,Y 380.105,Z 733.66,A -85,B 0,C 180,E1 11328.507,E2 11328.507} C_VEL
LIN {X 0,Y 380.54,Z 733.66,A -85,B 0,C 180,E1 11335.431,E2 11335.431} C_VEL
LIN {X 0,Y 380.857,Z 733.66,A -85,B 0,C 180,E1 11339.995,E2 11339.995} C_VEL
LIN {X 0,Y 380.477,Z 733.66,A -85,B 0,C 180,E1 11346.851,E2 11346.851} C_VEL
LIN {X 0,Y 380.122,Z 733.66,A -85,B 0,C 180,E1 11353.821,E2 11353.821} C_VEL
LIN {X 0,Y 379.836,Z 733.66,A -85,B 0,C 180,E1 11361.017,E2 11361.017} C_VEL
LIN {X 0,Y 379.544,Z 733.66,A -85,B 0,C 180,E1 11368.641,E2 11368.641} C_VEL
LIN {X 0,Y 379.408,Z 733.66,A -85,B 0,C 180,E1 11373.957,E2 11373.957} C_VEL
LIN {X 0,Y 379.231,Z 733.66,A -85,B 0,C 180,E1 11380.66,E2 11380.66} C_VEL
LIN {X 0,Y 379.484,Z 734.187,A -85,B 0,C 180,E1 11386.553,E2 11386.553} C_VEL
LIN {X 0,Y 385.188,Z 744.973,A -85,B 0,C 180,E1 11387.609,E2 11387.609} C_VEL
LIN {X 0,Y 394.843,Z 765.795,A -85,B 0,C 180,E1 11389.352,E2 11389.352} C_VEL
LIN {X 0,Y 411.277,Z 810.712,A -85,B 0,C 180,E1 11392.424,E2 11392.424} C_VEL
LIN {X 0,Y 407.278,Z 849.249,A -85,B 0,C 180,E1 11393.996,E2 11393.996} C_VEL
LIN {X 0,Y 402.257,Z 883.697,A -85,B 0,C 180,E1 11396.276,E2 11396.276} C_VEL
LIN {X 0,Y 396.255,Z 917.09,A -85,B 0,C 180,E1 11399.479,E2 11399.479} C_VEL
LIN {X 0,Y 390.642,Z 946.542,A -85,B 0,C 180,E1 11403.491,E2 11403.491} C_VEL
LIN {X 0,Y 386.167,Z 971.299,A -85,B 0,C 180,E1 11408.131,E2 11408.131} C_VEL
LIN {X 0,Y 383.097,Z 991.206,A -85,B 0,C 180,E1 11413.349,E2 11413.349} C_VEL
LIN {X 0,Y 381.673,Z 1004.814,A -85,B 0,C 180,E1 11418.559,E2 11418.559} C_VEL
LIN {X 0,Y 381.382,Z 1012.476,A -85,B 0,C 180,E1 11423.159,E2 11423.159} C_VEL
LIN {X 0,Y 381.262,Z 1016.168,A -85,B 0,C 180,E1 11427.748,E2 11427.748} C_VEL
LIN {X 0,Y 379.946,Z 1016.469,A -85,B 0,C 180,E1 11429.046,E2 11429.046} C_VEL
LIN {X 0,Y 373.493,Z 1015.638,A -85,B 0,C 180,E1 11432.599,E2 11432.599} C_VEL
LIN {X 0,Y 373.391,Z 1015.394,A -85,B 0,C 180,E1 11432.935,E2 11432.935} C_VEL
LIN {X 0,Y 373.543,Z 1010.493,A -85,B 0,C 180,E1 11438.156,E2 11438.156} C_VEL
LIN {X 0,Y 374.195,Z 1000.718,A -85,B 0,C 180,E1 11443.356,E2 11443.356} C_VEL
LIN {X 0,Y 376.164,Z 984.953,A -85,B 0,C 180,E1 11448.784,E2 11448.784} C_VEL
LIN {X 0,Y 379.856,Z 964.039,A -85,B 0,C 180,E1 11453.802,E2 11453.802} C_VEL
LIN {X 0,Y 384.896,Z 938.982,A -85,B 0,C 180,E1 11458.167,E2 11458.167} C_VEL
LIN {X 0,Y 390.91,Z 909.499,A -85,B 0,C 180,E1 11461.913,E2 11461.913} C_VEL
LIN {X 0,Y 396.739,Z 876.484,A -85,B 0,C 180,E1 11464.921,E2 11464.921} C_VEL
LIN {X 0,Y 402.055,Z 840.069,A -85,B 0,C 180,E1 11467.12,E2 11467.12} C_VEL
LIN {X 0,Y 404.654,Z 809.818,A -85,B 0,C 180,E1 11468.329,E2 11468.329} C_VEL
LIN {X 0,Y 395.338,Z 778.473,A -85,B 0,C 180,E1 11470.305,E2 11470.305} C_VEL
LIN {X 0,Y 388.622,Z 764.033,A -85,B 0,C 180,E1 11471.685,E2 11471.685} C_VEL
LIN {X 0,Y 385.326,Z 755.963,A -85,B 0,C 180,E1 11473.114,E2 11473.114} C_VEL
LIN {X 0,Y 380.241,Z 747.628,A -85,B 0,C 180,E1 11475.707,E2 11475.707} C_VEL
LIN {X 0,Y 376.786,Z 741.298,A -85,B 0,C 180,E1 11479.997,E2 11479.997} C_VEL
LIN {X 0,Y 376.786,Z 741.44,A -85,B 0,C 180,E1 11481.514,E2 11481.514} C_VEL
LIN {X 0,Y 379.713,Z 747.26,A -85,B 0,C 180,E1 11485.479,E2 11485.479} C_VEL
LIN {X 0,Y 384.736,Z 757.301,A -85,B 0,C 180,E1 11488.423,E2 11488.423} C_VEL
LIN {X 0,Y 391.101,Z 772.644,A -85,B 0,C 180,E1 11491.035,E2 11491.035} C_VEL
LIN {X 0,Y 393.839,Z 784.112,A -85,B 0,C 180,E1 11492.215,E2 11492.215} C_VEL
LIN {X 0,Y 391.251,Z 815.479,A -85,B 0,C 180,E1 11494.045,E2 11494.045} C_VEL
LIN {X 0,Y 388.06,Z 841.336,A -85,B 0,C 180,E1 11496.51,E2 11496.51} C_VEL
LIN {X 0,Y 384.517,Z 862.56,A -85,B 0,C 180,E1 11499.552,E2 11499.552} C_VEL
LIN {X 0,Y 381.126,Z 879.564,A -85,B 0,C 180,E1 11503.167,E2 11503.167} C_VEL
LIN {X 0,Y 378.376,Z 891.859,A -85,B 0,C 180,E1 11507.292,E2 11507.292} C_VEL
LIN {X 0,Y 376.818,Z 897.779,A -85,B 0,C 180,E1 11510.757,E2 11510.757} C_VEL
LIN {X 0,Y 375.785,Z 900.374,A -85,B 0,C 180,E1 11515.383,E2 11515.383} C_VEL
LIN {X 0,Y 375.507,Z 897.047,A -85,B 0,C 180,E1 11520.005,E2 11520.005} C_VEL
LIN {X 0,Y 375.92,Z 889.193,A -85,B 0,C 180,E1 11524.047,E2 11524.047} C_VEL
LIN {X 0,Y 376.945,Z 875.969,A -85,B 0,C 180,E1 11528.087,E2 11528.087} C_VEL
LIN {X 0,Y 378.67,Z 857.481,A -85,B 0,C 180,E1 11531.8,E2 11531.8} C_VEL
LIN {X 0,Y 380.791,Z 834.357,A -85,B 0,C 180,E1 11534.983,E2 11534.983} C_VEL
LIN {X 0,Y 382.841,Z 808.136,A -85,B 0,C 180,E1 11537.407,E2 11537.407} C_VEL
LIN {X 0,Y 384.315,Z 778.671,A -85,B 0,C 180,E1 11539.111,E2 11539.111} C_VEL
LIN {X 0,Y 371.867,Z 733.66,A -85,B 0,C 180,E1 11541.304,E2 11541.304} C_VEL
LIN {X 0,Y 371.646,Z 733.66,A -85,B 0,C 180,E1 11546.629,E2 11546.629} C_VEL
LIN {X 0,Y 371.497,Z 733.66,A -85,B 0,C 180,E1 11551.998,E2 11551.998} C_VEL
LIN {X 0,Y 371.284,Z 733.66,A -85,B 0,C 180,E1 11559.212,E2 11559.212} C_VEL
LIN {X 0,Y 371.38,Z 733.66,A -85,B 0,C 180,E1 11565.744,E2 11565.744} C_VEL
LIN {X 0,Y 373.892,Z 739.422,A -85,B 0,C 180,E1 11566.294,E2 11566.294} C_VEL
LIN {X 0,Y 392.591,Z 773.808,A -85,B 0,C 180,E1 11569.831,E2 11569.831} C_VEL
LIN {X 0,Y 404.249,Z 804.367,A -85,B 0,C 180,E1 11572.714,E2 11572.714} C_VEL
LIN {X 0,Y 399.579,Z 838.831,A -85,B 0,C 180,E1 11574.795,E2 11574.795} C_VEL
LIN {X 0,Y 393.94,Z 870.928,A -85,B 0,C 180,E1 11577.642,E2 11577.642} C_VEL
LIN {X 0,Y 387.663,Z 900.783,A -85,B 0,C 180,E1 11581.362,E2 11581.362} C_VEL
LIN {X 0,Y 382.141,Z 925.739,A -85,B 0,C 180,E1 11585.69,E2 11585.69} C_VEL
LIN {X 0,Y 377.803,Z 946.289,A -85,B 0,C 180,E1 11590.619,E2 11590.619} C_VEL
LIN {X 0,Y 375.102,Z 961.877,A -85,B 0,C 180,E1 11595.985,E2 11595.985} C_VEL
LIN {X 0,Y 373.678,Z 972.492,A -85,B 0,C 180,E1 11601.847,E2 11601.847} C_VEL
LIN {X 0,Y 373.326,Z 976.071,A -85,B 0,C 180,E1 11605.348,E2 11605.348} C_VEL
LIN {X 0,Y 373.319,Z 977.811,A -85,B 0,C 180,E1 11610,E2 11610} C_VEL
LIN {X 0,Y 373.491,Z 975.1,A -85,B 0,C 180,E1 11615.734,E2 11615.734} C_VEL
LIN {X 0,Y 374.365,Z 966.656,A -85,B 0,C 180,E1 11621.667,E2 11621.667} C_VEL
LIN {X 0,Y 376.421,Z 953.804,A -85,B 0,C 180,E1 11626.955,E2 11626.955} C_VEL
LIN {X 0,Y 380.268,Z 934.863,A -85,B 0,C 180,E1 11632.226,E2 11632.226} C_VEL
LIN {X 0,Y 385.361,Z 911.38,A -85,B 0,C 180,E1 11636.862,E2 11636.862} C_VEL
LIN {X 0,Y 391.202,Z 884.132,A -85,B 0,C 180,E1 11640.772,E2 11640.772} C_VEL
LIN {X 0,Y 397.279,Z 852.347,A -85,B 0,C 180,E1 11644.04,E2 11644.04} C_VEL
LIN {X 0,Y 402.688,Z 817.351,A -85,B 0,C 180,E1 11646.502,E2 11646.502} C_VEL
LIN {X 0,Y 403.824,Z 802.919,A -85,B 0,C 180,E1 11647.324,E2 11647.324} C_VEL
LIN {X 0,Y 392.033,Z 772.679,A -85,B 0,C 180,E1 11650.18,E2 11650.18} C_VEL
LIN {X 0,Y 373.304,Z 738.932,A -85,B 0,C 180,E1 11653.697,E2 11653.697} C_VEL
LIN {X 0,Y 371.315,Z 733.66,A -85,B 0,C 180,E1 11654.167,E2 11654.167} C_VEL
LIN {X 0,Y 371.298,Z 733.66,A -85,B 0,C 180,E1 11660.786,E2 11660.786} C_VEL
LIN {X 0,Y 371.5,Z 733.66,A -85,B 0,C 180,E1 11668.002,E2 11668.002} C_VEL
LIN {X 0,Y 371.766,Z 733.66,A -85,B 0,C 180,E1 11675.962,E2 11675.962} C_VEL
LIN {X 0,Y 371.995,Z 733.66,A -85,B 0,C 180,E1 11680.993,E2 11680.993} C_VEL
LIN {X 0,Y 372.163,Z 733.66,A -85,B 0,C 180,E1 11688.258,E2 11688.258} C_VEL
LIN {X 0,Y 372.629,Z 733.66,A -85,B 0,C 180,E1 11695.334,E2 11695.334} C_VEL
LIN {X 0,Y 372.956,Z 733.66,A -85,B 0,C 180,E1 11699.995,E2 11699.995} C_VEL
LIN {X 0,Y 372.549,Z 733.66,A -85,B 0,C 180,E1 11706.998,E2 11706.998} C_VEL
LIN {X 0,Y 372.178,Z 733.66,A -85,B 0,C 180,E1 11714.122,E2 11714.122} C_VEL
LIN {X 0,Y 371.86,Z 733.66,A -85,B 0,C 180,E1 11721.49,E2 11721.49} C_VEL
LIN {X 0,Y 371.674,Z 733.66,A -85,B 0,C 180,E1 11726.615,E2 11726.615} C_VEL
LIN {X 0,Y 371.499,Z 733.66,A -85,B 0,C 180,E1 11731.986,E2 11731.986} C_VEL
LIN {X 0,Y 371.285,Z 733.66,A -85,B 0,C 180,E1 11739.211,E2 11739.211} C_VEL
LIN {X 0,Y 371.408,Z 733.66,A -85,B 0,C 180,E1 11745.344,E2 11745.344} C_VEL
LIN {X 0,Y 373.941,Z 739.385,A -85,B 0,C 180,E1 11745.885,E2 11745.885} C_VEL
LIN {X 0,Y 386.135,Z 761.913,A -85,B 0,C 180,E1 11748.149,E2 11748.149} C_VEL
LIN {X 0,Y 403.321,Z 808.225,A -85,B 0,C 180,E1 11751.477,E2 11751.477} C_VEL
LIN {X 0,Y 404.643,Z 816.115,A -85,B 0,C 180,E1 11751.936,E2 11751.936} C_VEL
LIN {X 0,Y 400.397,Z 852.506,A -85,B 0,C 180,E1 11753.53,E2 11753.53} C_VEL
LIN {X 0,Y 394.916,Z 887.613,A -85,B 0,C 180,E1 11755.983,E2 11755.983} C_VEL
LIN {X 0,Y 388.668,Z 919.841,A -85,B 0,C 180,E1 11759.259,E2 11759.259} C_VEL
LIN {X 0,Y 382.955,Z 948.212,A -85,B 0,C 180,E1 11763.288,E2 11763.288} C_VEL
LIN {X 0,Y 378.132,Z 973.492,A -85,B 0,C 180,E1 11768.272,E2 11768.272} C_VEL
LIN {X 0,Y 375.1,Z 992.569,A -85,B 0,C 180,E1 11773.587,E2 11773.587} C_VEL
LIN {X 0,Y 373.737,Z 1005.582,A -85,B 0,C 180,E1 11778.905,E2 11778.905} C_VEL
LIN {X 0,Y 373.458,Z 1013.367,A -85,B 0,C 180,E1 11784.231,E2 11784.231} C_VEL
LIN {X 0,Y 373.405,Z 1016.271,A -85,B 0,C 180,E1 11790,E2 11790} C_VEL
LIN {X 0,Y 373.391,Z 1015.394,A -85,B 0,C 180,E1 11792.935,E2 11792.935} C_VEL
LIN {X 0,Y 370.848,Z 1014.072,A -85,B 0,C 180,E1 11794.909,E2 11794.909} C_VEL
LIN {X 0,Y 365.706,Z 1010.723,A -85,B 0,C 180,E1 11797.861,E2 11797.861} C_VEL
LIN {X 0,Y 365.648,Z 1010.258,A -85,B 0,C 180,E1 11798.2,E2 11798.2} C_VEL
LIN {X 0,Y 366.354,Z 1000.274,A -85,B 0,C 180,E1 11803.662,E2 11803.662} C_VEL
LIN {X 0,Y 368.527,Z 984.541,A -85,B 0,C 180,E1 11809.188,E2 11809.188} C_VEL
LIN {X 0,Y 372.438,Z 963.628,A -85,B 0,C 180,E1 11814.306,E2 11814.306} C_VEL
LIN {X 0,Y 377.776,Z 938.576,A -85,B 0,C 180,E1 11818.747,E2 11818.747} C_VEL
LIN {X 0,Y 383.909,Z 909.992,A -85,B 0,C 180,E1 11822.449,E2 11822.449} C_VEL
LIN {X 0,Y 390.216,Z 876.103,A -85,B 0,C 180,E1 11825.592,E2 11825.592} C_VEL
LIN {X 0,Y 395.741,Z 839.709,A -85,B 0,C 180,E1 11827.815,E2 11827.815} C_VEL
LIN {X 0,Y 398.279,Z 812.168,A -85,B 0,C 180,E1 11828.954,E2 11828.954} C_VEL
LIN {X 0,Y 389.835,Z 782.501,A -85,B 0,C 180,E1 11830.894,E2 11830.894} C_VEL
LIN {X 0,Y 384.669,Z 770.966,A -85,B 0,C 180,E1 11832.039,E2 11832.039} C_VEL
LIN {X 0,Y 382.082,Z 763.188,A -85,B 0,C 180,E1 11833.366,E2 11833.366} C_VEL
LIN {X 0,Y 378.128,Z 755.611,A -85,B 0,C 180,E1 11835.536,E2 11835.536} C_VEL
LIN {X 0,Y 374.262,Z 749.233,A -85,B 0,C 180,E1 11839.672,E2 11839.672} C_VEL
LIN {X 0,Y 374.133,Z 750.693,A -85,B 0,C 180,E1 11842.633,E2 11842.633} C_VEL
LIN {X 0,Y 377.103,Z 755.888,A -85,B 0,C 180,E1 11845.807,E2 11845.807} C_VEL
LIN {X 0,Y 381.595,Z 765.65,A -85,B 0,C 180,E1 11848.513,E2 11848.513} C_VEL
LIN {X 0,Y 386.788,Z 780.427,A -85,B 0,C 180,E1 11850.887,E2 11850.887} C_VEL
LIN {X 0,Y 387.729,Z 787.844,A -85,B 0,C 180,E1 11851.575,E2 11851.575} C_VEL
LIN {X 0,Y 384.825,Z 818.457,A -85,B 0,C 180,E1 11853.494,E2 11853.494} C_VEL
LIN {X 0,Y 381.168,Z 844.413,A -85,B 0,C 180,E1 11856.088,E2 11856.088} C_VEL
LIN {X 0,Y 377.096,Z 866.456,A -85,B 0,C 180,E1 11859.438,E2 11859.438} C_VEL
LIN {X 0,Y 373.233,Z 883.906,A -85,B 0,C 180,E1 11863.509,E2 11863.509} C_VEL
LIN {X 0,Y 370.481,Z 894.757,A -85,B 0,C 180,E1 11867.616,E2 11867.616} C_VEL
LIN {X 0,Y 369.158,Z 899.326,A -85,B 0,C 180,E1 11870.563,E2 11870.563} C_VEL
LIN {X 0,Y 368.034,Z 901.745,A -85,B 0,C 180,E1 11875.286,E2 11875.286} C_VEL
LIN {X 0,Y 367.696,Z 898.271,A -85,B 0,C 180,E1 11880.005,E2 11880.005} C_VEL
LIN {X 0,Y 368.115,Z 890.279,A -85,B 0,C 180,E1 11884.133,E2 11884.133} C_VEL
LIN {X 0,Y 369.305,Z 875.685,A -85,B 0,C 180,E1 11888.552,E2 11888.552} C_VEL
LIN {X 0,Y 371.159,Z 856.387,A -85,B 0,C 180,E1 11892.371,E2 11892.371} C_VEL
LIN {X 0,Y 373.379,Z 832.341,A -85,B 0,C 180,E1 11895.589,E2 11895.589} C_VEL
LIN {X 0,Y 375.584,Z 804.541,A -85,B 0,C 180,E1 11898.058,E2 11898.058} C_VEL
LIN {X 0,Y 376.243,Z 776.476,A -85,B 0,C 180,E1 11899.625,E2 11899.625} C_VEL
LIN {X 0,Y 363.899,Z 733.66,A -85,B 0,C 180,E1 11901.78,E2 11901.78} C_VEL
LIN {X 0,Y 363.655,Z 733.66,A -85,B 0,C 180,E1 11909.033,E2 11909.033} C_VEL
LIN {X 0,Y 363.382,Z 733.66,A -85,B 0,C 180,E1 11915.69,E2 11915.69} C_VEL
LIN {X 0,Y 363.394,Z 733.66,A -85,B 0,C 180,E1 11921.813,E2 11921.813} C_VEL
LIN {X 0,Y 363.408,Z 733.692,A -85,B 0,C 180,E1 11924.521,E2 11924.521} C_VEL
LIN {X 0,Y 365.837,Z 739.358,A -85,B 0,C 180,E1 11925.064,E2 11925.064} C_VEL
LIN {X 0,Y 384.265,Z 772.145,A -85,B 0,C 180,E1 11928.69,E2 11928.69} C_VEL
LIN {X 0,Y 396.648,Z 803.283,A -85,B 0,C 180,E1 11931.775,E2 11931.775} C_VEL
LIN {X 0,Y 397.395,Z 809.598,A -85,B 0,C 180,E1 11932.269,E2 11932.269} C_VEL
LIN {X 0,Y 392.385,Z 843.994,A -85,B 0,C 180,E1 11934.491,E2 11934.491} C_VEL
LIN {X 0,Y 386.43,Z 875.409,A -85,B 0,C 180,E1 11937.46,E2 11937.46} C_VEL
LIN {X 0,Y 380.05,Z 903.989,A -85,B 0,C 180,E1 11941.224,E2 11941.224} C_VEL
LIN {X 0,Y 374.094,Z 929.467,A -85,B 0,C 180,E1 11945.878,E2 11945.878} C_VEL
LIN {X 0,Y 369.816,Z 948.964,A -85,B 0,C 180,E1 11950.881,E2 11950.881} C_VEL
LIN {X 0,Y 367.121,Z 963.58,A -85,B 0,C 180,E1 11956.282,E2 11956.282} C_VEL
LIN {X 0,Y 365.84,Z 972.899,A -85,B 0,C 180,E1 11961.672,E2 11961.672} C_VEL
LIN {X 0,Y 365.342,Z 977.767,A -85,B 0,C 180,E1 11967.625,E2 11967.625} C_VEL
LIN {X 0,Y 365.419,Z 977.722,A -85,B 0,C 180,E1 11972.375,E2 11972.375} C_VEL
LIN {X 0,Y 365.839,Z 972.779,A -85,B 0,C 180,E1 11978.329,E2 11978.329} C_VEL
LIN {X 0,Y 367.334,Z 962.072,A -85,B 0,C 180,E1 11984.319,E2 11984.319} C_VEL
LIN {X 0,Y 370.421,Z 945.901,A -85,B 0,C 180,E1 11989.921,E2 11989.921} C_VEL
LIN {X 0,Y 374.941,Z 925.557,A -85,B 0,C 180,E1 11994.843,E2 11994.843} C_VEL
LIN {X 0,Y 381.176,Z 898.978,A -85,B 0,C 180,E1 11999.442,E2 11999.442} C_VEL
LIN {X 0,Y 387.676,Z 868.88,A -85,B 0,C 180,E1 12003.147,E2 12003.147} C_VEL
LIN {X 0,Y 393.501,Z 836.928,A -85,B 0,C 180,E1 12005.94,E2 12005.94} C_VEL
LIN {X 0,Y 397.441,Z 805.709,A -85,B 0,C 180,E1 12007.874,E2 12007.874} C_VEL
LIN {X 0,Y 385.645,Z 775.125,A -85,B 0,C 180,E1 12010.902,E2 12010.902} C_VEL
LIN {X 0,Y 367.934,Z 743.216,A -85,B 0,C 180,E1 12014.393,E2 12014.393} C_VEL
LIN {X 0,Y 363.379,Z 734.321,A -85,B 0,C 180,E1 12015.353,E2 12015.353} C_VEL
LIN {X 0,Y 363.396,Z 733.66,A -85,B 0,C 180,E1 12022.339,E2 12022.339} C_VEL
LIN {X 0,Y 363.625,Z 733.66,A -85,B 0,C 180,E1 12030.018,E2 12030.018} C_VEL
LIN {X 0,Y 363.908,Z 733.66,A -85,B 0,C 180,E1 12038.005,E2 12038.005} C_VEL
LIN {X 0,Y 364.145,Z 733.66,A -85,B 0,C 180,E1 12045.549,E2 12045.549} C_VEL
LIN {X 0,Y 364.678,Z 733.66,A -85,B 0,C 180,E1 12052.84,E2 12052.84} C_VEL
LIN {X 0,Y 365.054,Z 733.66,A -85,B 0,C 180,E1 12059.995,E2 12059.995} C_VEL
LIN {X 0,Y 364.649,Z 733.66,A -85,B 0,C 180,E1 12067.15,E2 12067.15} C_VEL
LIN {X 0,Y 364.234,Z 733.66,A -85,B 0,C 180,E1 12074.437,E2 12074.437} C_VEL
LIN {X 0,Y 363.878,Z 733.66,A -85,B 0,C 180,E1 12081.986,E2 12081.986} C_VEL
LIN {X 0,Y 363.637,Z 733.66,A -85,B 0,C 180,E1 12089.969,E2 12089.969} C_VEL
LIN {X 0,Y 363.383,Z 733.66,A -85,B 0,C 180,E1 12097.658,E2 12097.658} C_VEL
LIN {X 0,Y 363.45,Z 733.66,A -85,B 0,C 180,E1 12104.088,E2 12104.088} C_VEL
LIN {X 0,Y 365.994,Z 739.474,A -85,B 0,C 180,E1 12104.68,E2 12104.68} C_VEL
LIN {X 0,Y 380.741,Z 765.881,A -85,B 0,C 180,E1 12107.524,E2 12107.524} C_VEL
LIN {X 0,Y 397.146,Z 810.924,A -85,B 0,C 180,E1 12110.875,E2 12110.875} C_VEL
LIN {X 0,Y 398.204,Z 818.237,A -85,B 0,C 180,E1 12111.317,E2 12111.317} C_VEL
LIN {X 0,Y 393.675,Z 854.552,A -85,B 0,C 180,E1 12112.976,E2 12112.976} C_VEL
LIN {X 0,Y 387.897,Z 889.17,A -85,B 0,C 180,E1 12115.495,E2 12115.495} C_VEL
LIN {X 0,Y 381.505,Z 920.559,A -85,B 0,C 180,E1 12118.779,E2 12118.779} C_VEL
LIN {X 0,Y 375.473,Z 948.959,A -85,B 0,C 180,E1 12122.925,E2 12122.925} C_VEL
LIN {X 0,Y 370.562,Z 973.27,A -85,B 0,C 180,E1 12127.855,E2 12127.855} C_VEL
LIN {X 0,Y 367.335,Z 992.152,A -85,B 0,C 180,E1 12133.23,E2 12133.23} C_VEL
LIN {X 0,Y 365.871,Z 1005.169,A -85,B 0,C 180,E1 12138.663,E2 12138.663} C_VEL
LIN {X 0,Y 365.564,Z 1012.491,A -85,B 0,C 180,E1 12143.659,E2 12143.659} C_VEL
LIN {X 0,Y 365.491,Z 1015.349,A -85,B 0,C 180,E1 12147.625,E2 12147.625} C_VEL
LIN {X 0,Y 365.496,Z 1015.033,A -85,B 0,C 180,E1 12152.919,E2 12152.919} C_VEL
LIN {X 0,Y 365.648,Z 1010.258,A -85,B 0,C 180,E1 12158.2,E2 12158.2} C_VEL
LIN {X 0,Y 363.338,Z 1007.315,A -85,B 0,C 180,E1 12160.179,E2 12160.179} C_VEL
LIN {X 0,Y 358.452,Z 1001.757,A -85,B 0,C 180,E1 12163.113,E2 12163.113} C_VEL
LIN {X 0,Y 358.427,Z 1001.018,A -85,B 0,C 180,E1 12163.446,E2 12163.446} C_VEL
LIN {X 0,Y 360.463,Z 986.36,A -85,B 0,C 180,E1 12168.92,E2 12168.92} C_VEL
LIN {X 0,Y 364.299,Z 966.611,A -85,B 0,C 180,E1 12174.09,E2 12174.09} C_VEL
LIN {X 0,Y 370.261,Z 940.102,A -85,B 0,C 180,E1 12179.053,E2 12179.053} C_VEL
LIN {X 0,Y 376.748,Z 911.252,A -85,B 0,C 180,E1 12182.92,E2 12182.92} C_VEL
LIN {X 0,Y 383.36,Z 877.645,A -85,B 0,C 180,E1 12186.138,E2 12186.138} C_VEL
LIN {X 0,Y 389.147,Z 841.878,A -85,B 0,C 180,E1 12188.412,E2 12188.412} C_VEL
LIN {X 0,Y 392.064,Z 814.885,A -85,B 0,C 180,E1 12189.553,E2 12189.553} C_VEL
LIN {X 0,Y 384.217,Z 786.075,A -85,B 0,C 180,E1 12191.53,E2 12191.53} C_VEL
LIN {X 0,Y 380.443,Z 777.141,A -85,B 0,C 180,E1 12192.497,E2 12192.497} C_VEL
LIN {X 0,Y 378.187,Z 769.063,A -85,B 0,C 180,E1 12193.903,E2 12193.903} C_VEL
LIN {X 0,Y 373.909,Z 761.622,A -85,B 0,C 180,E1 12196.507,E2 12196.507} C_VEL
LIN {X 0,Y 371.652,Z 757.238,A -85,B 0,C 180,E1 12199.33,E2 12199.33} C_VEL
LIN {X 0,Y 371.273,Z 756.639,A -85,B 0,C 180,E1 12200.79,E2 12200.79} C_VEL
LIN {X 0,Y 372.868,Z 761.02,A -85,B 0,C 180,E1 12204.745,E2 12204.745} C_VEL
LIN {X 0,Y 376.554,Z 769.644,A -85,B 0,C 180,E1 12207.606,E2 12207.606} C_VEL
LIN {X 0,Y 381.244,Z 783.637,A -85,B 0,C 180,E1 12210.151,E2 12210.151} C_VEL
LIN {X 0,Y 381.919,Z 791.21,A -85,B 0,C 180,E1 12210.889,E2 12210.889} C_VEL
LIN {X 0,Y 378.499,Z 821.892,A -85,B 0,C 180,E1 12212.941,E2 12212.941} C_VEL
LIN {X 0,Y 374.383,Z 847.417,A -85,B 0,C 180,E1 12215.626,E2 12215.626} C_VEL
LIN {X 0,Y 370.052,Z 868.802,A -85,B 0,C 180,E1 12219.029,E2 12219.029} C_VEL
LIN {X 0,Y 365.901,Z 885.865,A -85,B 0,C 180,E1 12223.169,E2 12223.169} C_VEL
LIN {X 0,Y 362.951,Z 896.474,A -85,B 0,C 180,E1 12227.355,E2 12227.355} C_VEL
LIN {X 0,Y 361.501,Z 900.897,A -85,B 0,C 180,E1 12230.362,E2 12230.362} C_VEL
LIN {X 0,Y 360.277,Z 903.124,A -85,B 0,C 180,E1 12235.184,E2 12235.184} C_VEL
LIN {X 0,Y 359.915,Z 899.495,A -85,B 0,C 180,E1 12240.005,E2 12240.005} C_VEL
LIN {X 0,Y 360.309,Z 891.36,A -85,B 0,C 180,E1 12244.222,E2 12244.222} C_VEL
LIN {X 0,Y 361.575,Z 876.563,A -85,B 0,C 180,E1 12248.736,E2 12248.736} C_VEL
LIN {X 0,Y 363.48,Z 857.076,A -85,B 0,C 180,E1 12252.637,E2 12252.637} C_VEL
LIN {X 0,Y 365.803,Z 832.848,A -85,B 0,C 180,E1 12255.92,E2 12255.92} C_VEL
LIN {X 0,Y 368.108,Z 804.809,A -85,B 0,C 180,E1 12258.438,E2 12258.438} C_VEL
LIN {X 0,Y 368.719,Z 777.941,A -85,B 0,C 180,E1 12259.973,E2 12259.973} C_VEL
LIN {X 0,Y 355.923,Z 733.66,A -85,B 0,C 180,E1 12262.288,E2 12262.288} C_VEL
LIN {X 0,Y 355.745,Z 733.66,A -85,B 0,C 180,E1 12267.92,E2 12267.92} C_VEL
LIN {X 0,Y 355.475,Z 733.66,A -85,B 0,C 180,E1 12275.975,E2 12275.975} C_VEL
LIN {X 0,Y 355.459,Z 733.66,A -85,B 0,C 180,E1 12283.178,E2 12283.178} C_VEL
LIN {X 0,Y 357.793,Z 739.207,A -85,B 0,C 180,E1 12283.75,E2 12283.75} C_VEL
LIN {X 0,Y 376.883,Z 772.351,A -85,B 0,C 180,E1 12287.689,E2 12287.689} C_VEL
LIN {X 0,Y 389.691,Z 804.165,A -85,B 0,C 180,E1 12290.997,E2 12290.997} C_VEL
LIN {X 0,Y 391.009,Z 811.295,A -85,B 0,C 180,E1 12291.629,E2 12291.629} C_VEL
LIN {X 0,Y 385.706,Z 845.813,A -85,B 0,C 180,E1 12293.927,E2 12293.927} C_VEL
LIN {X 0,Y 379.315,Z 877.775,A -85,B 0,C 180,E1 12297.045,E2 12297.045} C_VEL
LIN {X 0,Y 372.752,Z 905.639,A -85,B 0,C 180,E1 12300.828,E2 12300.828} C_VEL
LIN {X 0,Y 366.547,Z 930.928,A -85,B 0,C 180,E1 12305.603,E2 12305.603} C_VEL
LIN {X 0,Y 361.823,Z 951.26,A -85,B 0,C 180,E1 12311.077,E2 12311.077} C_VEL
LIN {X 0,Y 359.083,Z 965.561,A -85,B 0,C 180,E1 12316.725,E2 12316.725} C_VEL
LIN {X 0,Y 357.825,Z 974.768,A -85,B 0,C 180,E1 12322.707,E2 12322.707} C_VEL
LIN {X 0,Y 357.452,Z 978.173,A -85,B 0,C 180,E1 12327.573,E2 12327.573} C_VEL
LIN {X 0,Y 357.527,Z 978.129,A -85,B 0,C 180,E1 12332.428,E2 12332.428} C_VEL
LIN {X 0,Y 357.984,Z 973.188,A -85,B 0,C 180,E1 12338.513,E2 12338.513} C_VEL
LIN {X 0,Y 359.612,Z 962.482,A -85,B 0,C 180,E1 12344.633,E2 12344.633} C_VEL
LIN {X 0,Y 362.933,Z 946.311,A -85,B 0,C 180,E1 12350.35,E2 12350.35} C_VEL
LIN {X 0,Y 367.773,Z 925.711,A -85,B 0,C 180,E1 12355.42,E2 12355.42} C_VEL
LIN {X 0,Y 374.243,Z 899.375,A -85,B 0,C 180,E1 12360.044,E2 12360.044} C_VEL
LIN {X 0,Y 381.051,Z 869.278,A -85,B 0,C 180,E1 12363.8,E2 12363.8} C_VEL
LIN {X 0,Y 387.133,Z 837.317,A -85,B 0,C 180,E1 12366.626,E2 12366.626} C_VEL
LIN {X 0,Y 390.832,Z 807.975,A -85,B 0,C 180,E1 12368.509,E2 12368.509} C_VEL
LIN {X 0,Y 379.301,Z 777.719,A -85,B 0,C 180,E1 12371.646,E2 12371.646} C_VEL
LIN {X 0,Y 361.441,Z 745.136,A -85,B 0,C 180,E1 12375.366,E2 12375.366} C_VEL
LIN {X 0,Y 355.568,Z 734.976,A -85,B 0,C 180,E1 12376.635,E2 12376.635} C_VEL
LIN {X 0,Y 355.437,Z 733.66,A -85,B 0,C 180,E1 12376.754,E2 12376.754} C_VEL
LIN {X 0,Y 355.483,Z 733.66,A -85,B 0,C 180,E1 12384.024,E2 12384.024} C_VEL
LIN {X 0,Y 355.758,Z 733.66,A -85,B 0,C 180,E1 12392.081,E2 12392.081} C_VEL
LIN {X 0,Y 356.095,Z 733.66,A -85,B 0,C 180,E1 12400.109,E2 12400.109} C_VEL
LIN {X 0,Y 356.317,Z 733.66,A -85,B 0,C 180,E1 12407.78,E2 12407.78} C_VEL
LIN {X 0,Y 356.839,Z 733.66,A -85,B 0,C 180,E1 12415.127,E2 12415.127} C_VEL
LIN {X 0,Y 357.164,Z 733.66,A -85,B 0,C 180,E1 12419.995,E2 12419.995} C_VEL
LIN {X 0,Y 356.716,Z 733.66,A -85,B 0,C 180,E1 12427.31,E2 12427.31} C_VEL
LIN {X 0,Y 356.287,Z 733.66,A -85,B 0,C 180,E1 12434.766,E2 12434.766} C_VEL
LIN {X 0,Y 355.934,Z 733.66,A -85,B 0,C 180,E1 12442.503,E2 12442.503} C_VEL
LIN {X 0,Y 355.756,Z 733.66,A -85,B 0,C 180,E1 12447.907,E2 12447.907} C_VEL
LIN {X 0,Y 355.478,Z 733.66,A -85,B 0,C 180,E1 12455.975,E2 12455.975} C_VEL
LIN {X 0,Y 355.461,Z 733.66,A -85,B 0,C 180,E1 12462.753,E2 12462.753} C_VEL
LIN {X 0,Y 358.001,Z 739.45,A -85,B 0,C 180,E1 12463.382,E2 12463.382} C_VEL
LIN {X 0,Y 374.999,Z 768.711,A -85,B 0,C 180,E1 12466.795,E2 12466.795} C_VEL
LIN {X 0,Y 390.569,Z 812.41,A -85,B 0,C 180,E1 12470.168,E2 12470.168} C_VEL
LIN {X 0,Y 391.792,Z 820.371,A -85,B 0,C 180,E1 12470.676,E2 12470.676} C_VEL
LIN {X 0,Y 386.815,Z 857.508,A -85,B 0,C 180,E1 12472.471,E2 12472.471} C_VEL
LIN {X 0,Y 380.866,Z 890.943,A -85,B 0,C 180,E1 12475.009,E2 12475.009} C_VEL
LIN {X 0,Y 374.099,Z 922.438,A -85,B 0,C 180,E1 12478.424,E2 12478.424} C_VEL
LIN {X 0,Y 367.753,Z 950.779,A -85,B 0,C 180,E1 12482.745,E2 12482.745} C_VEL
LIN {X 0,Y 362.957,Z 973.32,A -85,B 0,C 180,E1 12487.488,E2 12487.488} C_VEL
LIN {X 0,Y 359.584,Z 991.736,A -85,B 0,C 180,E1 12492.857,E2 12492.857} C_VEL
LIN {X 0,Y 358.014,Z 1004.756,A -85,B 0,C 180,E1 12498.411,E2 12498.411} C_VEL
LIN {X 0,Y 357.67,Z 1012.082,A -85,B 0,C 180,E1 12503.519,E2 12503.519} C_VEL
LIN {X 0,Y 357.593,Z 1014.942,A -85,B 0,C 180,E1 12507.573,E2 12507.573} C_VEL
LIN {X 0,Y 357.645,Z 1014.948,A -85,B 0,C 180,E1 12512.426,E2 12512.426} C_VEL
LIN {X 0,Y 357.748,Z 1010.067,A -85,B 0,C 180,E1 12518.213,E2 12518.213} C_VEL
LIN {X 0,Y 358.427,Z 1001.018,A -85,B 0,C 180,E1 12523.446,E2 12523.446} C_VEL
LIN {X 0,Y 355.216,Z 995.068,A -85,B 0,C 180,E1 12526.047,E2 12526.047} C_VEL
LIN {X 0,Y 352.406,Z 988.182,A -85,B 0,C 180,E1 12528.632,E2 12528.632} C_VEL
LIN {X 0,Y 356.47,Z 968.127,A -85,B 0,C 180,E1 12534.177,E2 12534.177} C_VEL
LIN {X 0,Y 362.286,Z 943.401,A -85,B 0,C 180,E1 12539.065,E2 12539.065} C_VEL
LIN {X 0,Y 369.451,Z 913.162,A -85,B 0,C 180,E1 12543.337,E2 12543.337} C_VEL
LIN {X 0,Y 376.286,Z 880.388,A -85,B 0,C 180,E1 12546.6,E2 12546.6} C_VEL
LIN {X 0,Y 382.578,Z 844.261,A -85,B 0,C 180,E1 12549.013,E2 12549.013} C_VEL
LIN {X 0,Y 385.537,Z 816.189,A -85,B 0,C 180,E1 12550.281,E2 12550.281} C_VEL
LIN {X 0,Y 379.089,Z 790.938,A -85,B 0,C 180,E1 12552.074,E2 12552.074} C_VEL
LIN {X 0,Y 376.169,Z 783.237,A -85,B 0,C 180,E1 12552.958,E2 12552.958} C_VEL
LIN {X 0,Y 374.292,Z 775.032,A -85,B 0,C 180,E1 12554.427,E2 12554.427} C_VEL
LIN {X 0,Y 371.677,Z 769.697,A -85,B 0,C 180,E1 12556.18,E2 12556.18} C_VEL
LIN {X 0,Y 368.936,Z 765.333,A -85,B 0,C 180,E1 12558.966,E2 12558.966} C_VEL
LIN {X 0,Y 368.318,Z 764.912,A -85,B 0,C 180,E1 12561.939,E2 12561.939} C_VEL
LIN {X 0,Y 370.106,Z 769.225,A -85,B 0,C 180,E1 12565.067,E2 12565.067} C_VEL
LIN {X 0,Y 373.422,Z 778.5,A -85,B 0,C 180,E1 12567.812,E2 12567.812} C_VEL
LIN {X 0,Y 376.757,Z 791.244,A -85,B 0,C 180,E1 12569.946,E2 12569.946} C_VEL
LIN {X 0,Y 372.342,Z 824.771,A -85,B 0,C 180,E1 12572.301,E2 12572.301} C_VEL
LIN {X 0,Y 368.058,Z 848.804,A -85,B 0,C 180,E1 12574.921,E2 12574.921} C_VEL
LIN {X 0,Y 363.448,Z 869.719,A -85,B 0,C 180,E1 12578.308,E2 12578.308} C_VEL
LIN {X 0,Y 359.196,Z 885.769,A -85,B 0,C 180,E1 12582.177,E2 12582.177} C_VEL
LIN {X 0,Y 355.86,Z 897.068,A -85,B 0,C 180,E1 12586.473,E2 12586.473} C_VEL
LIN {X 0,Y 353.86,Z 902.495,A -85,B 0,C 180,E1 12590.151,E2 12590.151} C_VEL
LIN {X 0,Y 352.529,Z 904.501,A -85,B 0,C 180,E1 12595.078,E2 12595.078} C_VEL
LIN {X 0,Y 352.1,Z 900.704,A -85,B 0,C 180,E1 12600.006,E2 12600.006} C_VEL
LIN {X 0,Y 352.511,Z 892.42,A -85,B 0,C 180,E1 12604.316,E2 12604.316} C_VEL
LIN {X 0,Y 353.843,Z 877.448,A -85,B 0,C 180,E1 12608.928,E2 12608.928} C_VEL
LIN {X 0,Y 355.808,Z 857.727,A -85,B 0,C 180,E1 12612.914,E2 12612.914} C_VEL
LIN {X 0,Y 358.246,Z 833.262,A -85,B 0,C 180,E1 12616.265,E2 12616.265} C_VEL
LIN {X 0,Y 360.575,Z 805.383,A -85,B 0,C 180,E1 12618.795,E2 12618.795} C_VEL
LIN {X 0,Y 361.235,Z 779.525,A -85,B 0,C 180,E1 12620.311,E2 12620.311} C_VEL
LIN {X 0,Y 347.959,Z 733.66,A -85,B 0,C 180,E1 12622.837,E2 12622.837} C_VEL
LIN {X 0,Y 347.67,Z 733.66,A -85,B 0,C 180,E1 12629.426,E2 12629.426} C_VEL
LIN {X 0,Y 347.527,Z 733.66,A -85,B 0,C 180,E1 12634.503,E2 12634.503} C_VEL
LIN {X 0,Y 347.412,Z 733.66,A -85,B 0,C 180,E1 12641.711,E2 12641.711} C_VEL
LIN {X 0,Y 349.939,Z 739.365,A -85,B 0,C 180,E1 12642.384,E2 12642.384} C_VEL
LIN {X 0,Y 369.33,Z 772.199,A -85,B 0,C 180,E1 12646.589,E2 12646.589} C_VEL
LIN {X 0,Y 382.219,Z 803.384,A -85,B 0,C 180,E1 12650.001,E2 12650.001} C_VEL
LIN {X 0,Y 384.681,Z 812.992,A -85,B 0,C 180,E1 12650.968,E2 12650.968} C_VEL
LIN {X 0,Y 378.995,Z 847.856,A -85,B 0,C 180,E1 12653.362,E2 12653.362} C_VEL
LIN {X 0,Y 372.398,Z 879.336,A -85,B 0,C 180,E1 12656.518,E2 12656.518} C_VEL
LIN {X 0,Y 365.387,Z 907.711,A -85,B 0,C 180,E1 12660.487,E2 12660.487} C_VEL
LIN {X 0,Y 358.909,Z 932.623,A -85,B 0,C 180,E1 12665.381,E2 12665.381} C_VEL
LIN {X 0,Y 354.259,Z 951.668,A -85,B 0,C 180,E1 12670.657,E2 12670.657} C_VEL
LIN {X 0,Y 351.285,Z 966.248,A -85,B 0,C 180,E1 12676.562,E2 12676.562} C_VEL
LIN {X 0,Y 349.962,Z 975.175,A -85,B 0,C 180,E1 12682.543,E2 12682.543} C_VEL
LIN {X 0,Y 349.561,Z 978.58,A -85,B 0,C 180,E1 12687.518,E2 12687.518} C_VEL
LIN {X 0,Y 349.635,Z 978.536,A -85,B 0,C 180,E1 12692.482,E2 12692.482} C_VEL
LIN {X 0,Y 349.962,Z 975.082,A -85,B 0,C 180,E1 12697.458,E2 12697.458} C_VEL
LIN {X 0,Y 351.344,Z 966.044,A -85,B 0,C 180,E1 12703.44,E2 12703.44} C_VEL
LIN {X 0,Y 354.307,Z 951.379,A -85,B 0,C 180,E1 12709.341,E2 12709.341} C_VEL
LIN {X 0,Y 359.328,Z 930.942,A -85,B 0,C 180,E1 12714.921,E2 12714.921} C_VEL
LIN {X 0,Y 365.91,Z 905.479,A -85,B 0,C 180,E1 12719.772,E2 12719.772} C_VEL
LIN {X 0,Y 372.826,Z 877.013,A -85,B 0,C 180,E1 12723.666,E2 12723.666} C_VEL
LIN {X 0,Y 379.745,Z 843.585,A -85,B 0,C 180,E1 12726.89,E2 12726.89} C_VEL
LIN {X 0,Y 384.408,Z 810.544,A -85,B 0,C 180,E1 12729.127,E2 12729.127} C_VEL
LIN {X 0,Y 372.761,Z 779.7,A -85,B 0,C 180,E1 12732.479,E2 12732.479} C_VEL
LIN {X 0,Y 356.077,Z 749.307,A -85,B 0,C 180,E1 12736.135,E2 12736.135} C_VEL
LIN {X 0,Y 347.535,Z 735.002,A -85,B 0,C 180,E1 12738.069,E2 12738.069} C_VEL
LIN {X 0,Y 347.397,Z 733.66,A -85,B 0,C 180,E1 12738.21,E2 12738.21} C_VEL
LIN {X 0,Y 347.564,Z 733.66,A -85,B 0,C 180,E1 12745.863,E2 12745.863} C_VEL
LIN {X 0,Y 347.736,Z 733.66,A -85,B 0,C 180,E1 12751.378,E2 12751.378} C_VEL
LIN {X 0,Y 348.148,Z 733.66,A -85,B 0,C 180,E1 12759.635,E2 12759.635} C_VEL
LIN {X 0,Y 348.263,Z 733.66,A -85,B 0,C 180,E1 12764.874,E2 12764.874} C_VEL
LIN {X 0,Y 348.798,Z 733.66,A -85,B 0,C 180,E1 12772.512,E2 12772.512} C_VEL
LIN {X 0,Y 349.262,Z 733.66,A -85,B 0,C 180,E1 12779.994,E2 12779.994} C_VEL
LIN {X 0,Y 348.786,Z 733.66,A -85,B 0,C 180,E1 12787.477,E2 12787.477} C_VEL
LIN {X 0,Y 348.34,Z 733.66,A -85,B 0,C 180,E1 12795.111,E2 12795.111} C_VEL
LIN {X 0,Y 348.135,Z 733.66,A -85,B 0,C 180,E1 12800.354,E2 12800.354} C_VEL
LIN {X 0,Y 347.738,Z 733.66,A -85,B 0,C 180,E1 12808.609,E2 12808.609} C_VEL
LIN {X 0,Y 347.562,Z 733.66,A -85,B 0,C 180,E1 12814.485,E2 12814.485} C_VEL
LIN {X 0,Y 347.624,Z 734.214,A -85,B 0,C 180,E1 12821.399,E2 12821.399} C_VEL
LIN {X 0,Y 350.297,Z 739.606,A -85,B 0,C 180,E1 12822.049,E2 12822.049} C_VEL
LIN {X 0,Y 369.369,Z 771.84,A -85,B 0,C 180,E1 12826.059,E2 12826.059} C_VEL
LIN {X 0,Y 383.97,Z 813.607,A -85,B 0,C 180,E1 12829.417,E2 12829.417} C_VEL
LIN {X 0,Y 385.403,Z 822.887,A -85,B 0,C 180,E1 12830.039,E2 12830.039} C_VEL
LIN {X 0,Y 380.338,Z 858.19,A -85,B 0,C 180,E1 12831.808,E2 12831.808} C_VEL
LIN {X 0,Y 374.171,Z 891.255,A -85,B 0,C 180,E1 12834.37,E2 12834.37} C_VEL
LIN {X 0,Y 366.964,Z 923.19,A -85,B 0,C 180,E1 12837.911,E2 12837.911} C_VEL
LIN {X 0,Y 360.149,Z 951.96,A -85,B 0,C 180,E1 12842.454,E2 12842.454} C_VEL
LIN {X 0,Y 355.077,Z 974.649,A -85,B 0,C 180,E1 12847.432,E2 12847.432} C_VEL
LIN {X 0,Y 351.586,Z 993.098,A -85,B 0,C 180,E1 12853.101,E2 12853.101} C_VEL
LIN {X 0,Y 350.083,Z 1005.498,A -85,B 0,C 180,E1 12858.777,E2 12858.777} C_VEL
LIN {X 0,Y 349.741,Z 1012.82,A -85,B 0,C 180,E1 12864.599,E2 12864.599} C_VEL
LIN {X 0,Y 349.748,Z 1015.052,A -85,B 0,C 180,E1 12870,E2 12870} C_VEL
LIN {X 0,Y 349.778,Z 1012.781,A -85,B 0,C 180,E1 12875.465,E2 12875.465} C_VEL
LIN {X 0,Y 350.118,Z 1005.507,A -85,B 0,C 180,E1 12881.221,E2 12881.221} C_VEL
LIN {X 0,Y 351.671,Z 993.12,A -85,B 0,C 180,E1 12886.894,E2 12886.894} C_VEL
LIN {X 0,Y 352.406,Z 988.182,A -85,B 0,C 180,E1 12888.632,E2 12888.632} C_VEL
LIN {X 0,Y 350.107,Z 980.468,A -85,B 0,C 180,E1 12891.171,E2 12891.171} C_VEL
LIN {X 0,Y 348.139,Z 971.976,A -85,B 0,C 180,E1 12893.677,E2 12893.677} C_VEL
LIN {X 0,Y 354.146,Z 947.119,A -85,B 0,C 180,E1 12898.983,E2 12898.983} C_VEL
LIN {X 0,Y 361.118,Z 919.391,A -85,B 0,C 180,E1 12903.208,E2 12903.208} C_VEL
LIN {X 0,Y 368.442,Z 886.975,A -85,B 0,C 180,E1 12906.744,E2 12906.744} C_VEL
LIN {X 0,Y 375.305,Z 851.186,A -85,B 0,C 180,E1 12909.356,E2 12909.356} C_VEL
LIN {X 0,Y 379.409,Z 818.93,A -85,B 0,C 180,E1 12910.922,E2 12910.922} C_VEL
LIN {X 0,Y 373.576,Z 794.842,A -85,B 0,C 180,E1 12912.713,E2 12912.713} C_VEL
LIN {X 0,Y 371.596,Z 787.591,A -85,B 0,C 180,E1 12913.694,E2 12913.694} C_VEL
LIN {X 0,Y 370.028,Z 780.447,A -85,B 0,C 180,E1 12915.148,E2 12915.148} C_VEL
LIN {X 0,Y 367.496,Z 775.692,A -85,B 0,C 180,E1 12917.087,E2 12917.087} C_VEL
LIN {X 0,Y 366.188,Z 773.405,A -85,B 0,C 180,E1 12918.591,E2 12918.591} C_VEL
LIN {X 0,Y 365.326,Z 772.338,A -85,B 0,C 180,E1 12921.948,E2 12921.948} C_VEL
LIN {X 0,Y 366.886,Z 777.27,A -85,B 0,C 180,E1 12925.179,E2 12925.179} C_VEL
LIN {X 0,Y 369.866,Z 786.806,A -85,B 0,C 180,E1 12927.856,E2 12927.856} C_VEL
LIN {X 0,Y 371.291,Z 795.708,A -85,B 0,C 180,E1 12929.239,E2 12929.239} C_VEL
LIN {X 0,Y 366.332,Z 827.711,A -85,B 0,C 180,E1 12931.628,E2 12931.628} C_VEL
LIN {X 0,Y 361.38,Z 852.224,A -85,B 0,C 180,E1 12934.444,E2 12934.444} C_VEL
LIN {X 0,Y 356.095,Z 873.745,A -85,B 0,C 180,E1 12938.165,E2 12938.165} C_VEL
LIN {X 0,Y 351.357,Z 889.915,A -85,B 0,C 180,E1 12942.45,E2 12942.45} C_VEL
LIN {X 0,Y 347.551,Z 901.008,A -85,B 0,C 180,E1 12947.425,E2 12947.425} C_VEL
LIN {X 0,Y 345.397,Z 905.728,A -85,B 0,C 180,E1 12952.449,E2 12952.449} C_VEL
LIN {X 0,Y 344.362,Z 904.63,A -85,B 0,C 180,E1 12957.486,E2 12957.486} C_VEL
LIN {X 0,Y 344.456,Z 897.664,A -85,B 0,C 180,E1 12962.525,E2 12962.525} C_VEL
LIN {X 0,Y 345.372,Z 885.183,A -85,B 0,C 180,E1 12967.246,E2 12967.246} C_VEL
LIN {X 0,Y 347.185,Z 867.363,A -85,B 0,C 180,E1 12971.551,E2 12971.551} C_VEL
LIN {X 0,Y 349.593,Z 844.956,A -85,B 0,C 180,E1 12975.227,E2 12975.227} C_VEL
LIN {X 0,Y 352.091,Z 818.342,A -85,B 0,C 180,E1 12978.165,E2 12978.165} C_VEL
LIN {X 0,Y 354.101,Z 788.675,A -85,B 0,C 180,E1 12980.249,E2 12980.249} C_VEL
LIN {X 0,Y 352.647,Z 776.741,A -85,B 0,C 180,E1 12980.92,E2 12980.92} C_VEL
LIN {X 0,Y 339.972,Z 733.66,A -85,B 0,C 180,E1 12983.462,E2 12983.462} C_VEL
LIN {X 0,Y 339.773,Z 733.66,A -85,B 0,C 180,E1 12989.357,E2 12989.357} C_VEL
LIN {X 0,Y 339.442,Z 733.66,A -85,B 0,C 180,E1 12996.593,E2 12996.593} C_VEL
LIN {X 0,Y 339.47,Z 734.202,A -85,B 0,C 180,E1 13000.228,E2 13000.228} C_VEL
LIN {X 0,Y 342.324,Z 739.707,A -85,B 0,C 180,E1 13000.968,E2 13000.968} C_VEL
LIN {X 0,Y 361.618,Z 771.805,A -85,B 0,C 180,E1 13005.385,E2 13005.385} C_VEL
LIN {X 0,Y 374.641,Z 802.43,A -85,B 0,C 180,E1 13008.933,E2 13008.933} C_VEL
LIN {X 0,Y 378.267,Z 815.463,A -85,B 0,C 180,E1 13010.335,E2 13010.335} C_VEL
LIN {X 0,Y 372.323,Z 849.899,A -85,B 0,C 180,E1 13012.778,E2 13012.778} C_VEL
LIN {X 0,Y 365.299,Z 881.776,A -85,B 0,C 180,E1 13016.076,E2 13016.076} C_VEL
LIN {X 0,Y 358.034,Z 909.737,A -85,B 0,C 180,E1 13020.131,E2 13020.131} C_VEL
LIN {X 0,Y 351.205,Z 934.638,A -85,B 0,C 180,E1 13025.229,E2 13025.229} C_VEL
LIN {X 0,Y 346.238,Z 954.053,A -85,B 0,C 180,E1 13030.886,E2 13030.886} C_VEL
LIN {X 0,Y 343.444,Z 967.116,A -85,B 0,C 180,E1 13036.482,E2 13036.482} C_VEL
LIN {X 0,Y 342.099,Z 975.583,A -85,B 0,C 180,E1 13042.37,E2 13042.37} C_VEL
LIN {X 0,Y 341.698,Z 978.985,A -85,B 0,C 180,E1 13047.461,E2 13047.461} C_VEL
LIN {X 0,Y 341.769,Z 978.942,A -85,B 0,C 180,E1 13052.54,E2 13052.54} C_VEL
LIN {X 0,Y 342.315,Z 974.005,A -85,B 0,C 180,E1 13058.906,E2 13058.906} C_VEL
LIN {X 0,Y 344.214,Z 963.303,A -85,B 0,C 180,E1 13065.303,E2 13065.303} C_VEL
LIN {X 0,Y 348.07,Z 946.801,A -85,B 0,C 180,E1 13071.365,E2 13071.365} C_VEL
LIN {X 0,Y 353.653,Z 925.691,A -85,B 0,C 180,E1 13076.714,E2 13076.714} C_VEL
LIN {X 0,Y 360.763,Z 899.163,A -85,B 0,C 180,E1 13081.466,E2 13081.466} C_VEL
LIN {X 0,Y 367.961,Z 870.076,A -85,B 0,C 180,E1 13085.175,E2 13085.175} C_VEL
LIN {X 0,Y 374.536,Z 838.303,A -85,B 0,C 180,E1 13088.051,E2 13088.051} C_VEL
LIN {X 0,Y 377.973,Z 813.018,A -85,B 0,C 180,E1 13089.781,E2 13089.781} C_VEL
LIN {X 0,Y 366.298,Z 781.706,A -85,B 0,C 180,E1 13093.34,E2 13093.34} C_VEL
LIN {X 0,Y 349.181,Z 750.554,A -85,B 0,C 180,E1 13097.299,E2 13097.299} C_VEL
LIN {X 0,Y 339.668,Z 735.358,A -85,B 0,C 180,E1 13099.571,E2 13099.571} C_VEL
LIN {X 0,Y 339.481,Z 733.66,A -85,B 0,C 180,E1 13099.698,E2 13099.698} C_VEL
LIN {X 0,Y 339.694,Z 733.66,A -85,B 0,C 180,E1 13107.874,E2 13107.874} C_VEL
LIN {X 0,Y 339.859,Z 733.66,A -85,B 0,C 180,E1 13113.539,E2 13113.539} C_VEL
LIN {X 0,Y 340.17,Z 733.66,A -85,B 0,C 180,E1 13119.182,E2 13119.182} C_VEL
LIN {X 0,Y 340.428,Z 733.66,A -85,B 0,C 180,E1 13127.146,E2 13127.146} C_VEL
LIN {X 0,Y 341.017,Z 733.66,A -85,B 0,C 180,E1 13134.9,E2 13134.9} C_VEL
LIN {X 0,Y 341.374,Z 733.66,A -85,B 0,C 180,E1 13139.994,E2 13139.994} C_VEL
LIN {X 0,Y 340.849,Z 733.66,A -85,B 0,C 180,E1 13147.652,E2 13147.652} C_VEL
LIN {X 0,Y 340.412,Z 733.66,A -85,B 0,C 180,E1 13155.471,E2 13155.471} C_VEL
LIN {X 0,Y 340.15,Z 733.66,A -85,B 0,C 180,E1 13160.854,E2 13160.854} C_VEL
LIN {X 0,Y 339.802,Z 733.66,A -85,B 0,C 180,E1 13169.341,E2 13169.341} C_VEL
LIN {X 0,Y 339.454,Z 733.66,A -85,B 0,C 180,E1 13176.594,E2 13176.594} C_VEL
LIN {X 0,Y 339.552,Z 734.37,A -85,B 0,C 180,E1 13179.849,E2 13179.849} C_VEL
LIN {X 0,Y 342.346,Z 739.648,A -85,B 0,C 180,E1 13180.567,E2 13180.567} C_VEL
LIN {X 0,Y 362.111,Z 772.302,A -85,B 0,C 180,E1 13184.964,E2 13184.964} C_VEL
LIN {X 0,Y 374.124,Z 803.711,A -85,B 0,C 180,E1 13187.707,E2 13187.707} C_VEL
LIN {X 0,Y 379.216,Z 823.656,A -85,B 0,C 180,E1 13189.317,E2 13189.317} C_VEL
LIN {X 0,Y 373.907,Z 858.871,A -85,B 0,C 180,E1 13191.122,E2 13191.122} C_VEL
LIN {X 0,Y 367.44,Z 891.85,A -85,B 0,C 180,E1 13193.733,E2 13193.733} C_VEL
LIN {X 0,Y 359.79,Z 924.25,A -85,B 0,C 180,E1 13197.425,E2 13197.425} C_VEL
LIN {X 0,Y 352.976,Z 951.547,A -85,B 0,C 180,E1 13201.845,E2 13201.845} C_VEL
LIN {X 0,Y 347.603,Z 974.234,A -85,B 0,C 180,E1 13206.919,E2 13206.919} C_VEL
LIN {X 0,Y 343.836,Z 992.681,A -85,B 0,C 180,E1 13212.708,E2 13212.708} C_VEL
LIN {X 0,Y 342.225,Z 1005.086,A -85,B 0,C 180,E1 13218.516,E2 13218.516} C_VEL
LIN {X 0,Y 341.82,Z 1011.676,A -85,B 0,C 180,E1 13223.642,E2 13223.642} C_VEL
LIN {X 0,Y 341.82,Z 1014.129,A -85,B 0,C 180,E1 13227.461,E2 13227.461} C_VEL
LIN {X 0,Y 341.871,Z 1014.135,A -85,B 0,C 180,E1 13232.538,E2 13232.538} C_VEL
LIN {X 0,Y 341.922,Z 1010.435,A -85,B 0,C 180,E1 13237.634,E2 13237.634} C_VEL
LIN {X 0,Y 342.66,Z 1001.191,A -85,B 0,C 180,E1 13243.603,E2 13243.603} C_VEL
LIN {X 0,Y 344.989,Z 986.505,A -85,B 0,C 180,E1 13249.478,E2 13249.478} C_VEL
LIN {X 0,Y 348.139,Z 971.976,A -85,B 0,C 180,E1 13253.677,E2 13253.677} C_VEL
LIN {X 0,Y 346.585,Z 962.79,A -85,B 0,C 180,E1 13256.129,E2 13256.129} C_VEL
LIN {X 0,Y 345.475,Z 952.678,A -85,B 0,C 180,E1 13258.494,E2 13258.494} C_VEL
LIN {X 0,Y 352.791,Z 925.141,A -85,B 0,C 180,E1 13263.093,E2 13263.093} C_VEL
LIN {X 0,Y 360.646,Z 893.049,A -85,B 0,C 180,E1 13266.883,E2 13266.883} C_VEL
LIN {X 0,Y 367.806,Z 858.685,A -85,B 0,C 180,E1 13269.647,E2 13269.647} C_VEL
LIN {X 0,Y 373.277,Z 821.272,A -85,B 0,C 180,E1 13271.607,E2 13271.607} C_VEL
LIN {X 0,Y 367.989,Z 798.542,A -85,B 0,C 180,E1 13273.383,E2 13273.383} C_VEL
LIN {X 0,Y 366.47,Z 787.365,A -85,B 0,C 180,E1 13275.394,E2 13275.394} C_VEL
LIN {X 0,Y 363.391,Z 781.394,A -85,B 0,C 180,E1 13278.201,E2 13278.201} C_VEL
LIN {X 0,Y 362.225,Z 779.413,A -85,B 0,C 180,E1 13281.181,E2 13281.181} C_VEL
LIN {X 0,Y 363.252,Z 783.674,A -85,B 0,C 180,E1 13284.727,E2 13284.727} C_VEL
LIN {X 0,Y 365.624,Z 792.949,A -85,B 0,C 180,E1 13287.437,E2 13287.437} C_VEL
LIN {X 0,Y 366.401,Z 798.184,A -85,B 0,C 180,E1 13288.347,E2 13288.347} C_VEL
LIN {X 0,Y 360.434,Z 830.984,A -85,B 0,C 180,E1 13290.949,E2 13290.949} C_VEL
LIN {X 0,Y 354.926,Z 855.327,A -85,B 0,C 180,E1 13293.891,E2 13293.891} C_VEL
LIN {X 0,Y 349.184,Z 876.346,A -85,B 0,C 180,E1 13297.71,E2 13297.71} C_VEL
LIN {X 0,Y 344.119,Z 892.016,A -85,B 0,C 180,E1 13302.069,E2 13302.069} C_VEL
LIN {X 0,Y 340.455,Z 901.789,A -85,B 0,C 180,E1 13306.505,E2 13306.505} C_VEL
LIN {X 0,Y 338.601,Z 905.748,A -85,B 0,C 180,E1 13309.703,E2 13309.703} C_VEL
LIN {X 0,Y 337.032,Z 907.277,A -85,B 0,C 180,E1 13314.851,E2 13314.851} C_VEL
LIN {X 0,Y 336.48,Z 903.102,A -85,B 0,C 180,E1 13320.006,E2 13320.006} C_VEL
LIN {X 0,Y 337,Z 892.782,A -85,B 0,C 180,E1 13325.161,E2 13325.161} C_VEL
LIN {X 0,Y 338.477,Z 877.761,A -85,B 0,C 180,E1 13329.662,E2 13329.662} C_VEL
LIN {X 0,Y 340.731,Z 856.952,A -85,B 0,C 180,E1 13333.824,E2 13333.824} C_VEL
LIN {X 0,Y 343.238,Z 832.45,A -85,B 0,C 180,E1 13337.162,E2 13337.162} C_VEL
LIN {X 0,Y 345.719,Z 804.282,A -85,B 0,C 180,E1 13339.713,E2 13339.713} C_VEL
LIN {X 0,Y 346.128,Z 782.147,A -85,B 0,C 180,E1 13341.052,E2 13341.052} C_VEL
LIN {X 0,Y 332.012,Z 733.66,A -85,B 0,C 180,E1 13343.982,E2 13343.982} C_VEL
LIN {X 0,Y 331.793,Z 733.66,A -85,B 0,C 180,E1 13350.135,E2 13350.135} C_VEL
LIN {X 0,Y 331.55,Z 733.66,A -85,B 0,C 180,E1 13358.55,E2 13358.55} C_VEL
LIN {X 0,Y 333.836,Z 739.242,A -85,B 0,C 180,E1 13359.231,E2 13359.231} C_VEL
LIN {X 0,Y 350.379,Z 765.283,A -85,B 0,C 180,E1 13363.271,E2 13363.271} C_VEL
LIN {X 0,Y 364.223,Z 793.679,A -85,B 0,C 180,E1 13366.885,E2 13366.885} C_VEL
LIN {X 0,Y 371.899,Z 817.84,A -85,B 0,C 180,E1 13369.68,E2 13369.68} C_VEL
LIN {X 0,Y 365.818,Z 851.353,A -85,B 0,C 180,E1 13372.121,E2 13372.121} C_VEL
LIN {X 0,Y 358.427,Z 883.358,A -85,B 0,C 180,E1 13375.511,E2 13375.511} C_VEL
LIN {X 0,Y 350.773,Z 911.31,A -85,B 0,C 180,E1 13379.693,E2 13379.693} C_VEL
LIN {X 0,Y 344.028,Z 934.79,A -85,B 0,C 180,E1 13384.608,E2 13384.608} C_VEL
LIN {X 0,Y 338.846,Z 953.847,A -85,B 0,C 180,E1 13390.231,E2 13390.231} C_VEL
LIN {X 0,Y 335.695,Z 967.524,A -85,B 0,C 180,E1 13396.164,E2 13396.164} C_VEL
LIN {X 0,Y 334.247,Z 975.99,A -85,B 0,C 180,E1 13402.19,E2 13402.19} C_VEL
LIN {X 0,Y 333.806,Z 979.392,A -85,B 0,C 180,E1 13407.401,E2 13407.401} C_VEL
LIN {X 0,Y 333.877,Z 979.349,A -85,B 0,C 180,E1 13412.6,E2 13412.6} C_VEL
LIN {X 0,Y 334.47,Z 974.414,A -85,B 0,C 180,E1 13419.117,E2 13419.117} C_VEL
LIN {X 0,Y 336.537,Z 963.713,A -85,B 0,C 180,E1 13425.661,E2 13425.661} C_VEL
LIN {X 0,Y 340.645,Z 947.211,A -85,B 0,C 180,E1 13431.855,E2 13431.855} C_VEL
LIN {X 0,Y 346.527,Z 926.101,A -85,B 0,C 180,E1 13437.309,E2 13437.309} C_VEL
LIN {X 0,Y 354,Z 899.567,A -85,B 0,C 180,E1 13442.139,E2 13442.139} C_VEL
LIN {X 0,Y 361.485,Z 870.476,A -85,B 0,C 180,E1 13445.902,E2 13445.902} C_VEL
LIN {X 0,Y 368.353,Z 838.611,A -85,B 0,C 180,E1 13448.816,E2 13448.816} C_VEL
LIN {X 0,Y 371.667,Z 815.805,A -85,B 0,C 180,E1 13450.411,E2 13450.411} C_VEL
LIN {X 0,Y 360.332,Z 784.829,A -85,B 0,C 180,E1 13454.093,E2 13454.093} C_VEL
LIN {X 0,Y 344.347,Z 755.309,A -85,B 0,C 180,E1 13458.04,E2 13458.04} C_VEL
LIN {X 0,Y 333.271,Z 738.582,A -85,B 0,C 180,E1 13460.784,E2 13460.784} C_VEL
LIN {X 0,Y 331.584,Z 733.66,A -85,B 0,C 180,E1 13461.368,E2 13461.368} C_VEL
LIN {X 0,Y 331.799,Z 733.66,A -85,B 0,C 180,E1 13469.865,E2 13469.865} C_VEL
LIN {X 0,Y 332.004,Z 733.66,A -85,B 0,C 180,E1 13475.797,E2 13475.797} C_VEL
LIN {X 0,Y 332.332,Z 733.66,A -85,B 0,C 180,E1 13483.09,E2 13483.09} C_VEL
LIN {X 0,Y 332.654,Z 733.66,A -85,B 0,C 180,E1 13489.505,E2 13489.505} C_VEL
LIN {X 0,Y 333.361,Z 733.66,A -85,B 0,C 180,E1 13497.391,E2 13497.391} C_VEL
LIN {X 0,Y 333.353,Z 733.66,A -85,B 0,C 180,E1 13502.597,E2 13502.597} C_VEL
LIN {X 0,Y 332.739,Z 733.66,A -85,B 0,C 180,E1 13510.481,E2 13510.481} C_VEL
LIN {X 0,Y 332.334,Z 733.66,A -85,B 0,C 180,E1 13518.59,E2 13518.59} C_VEL
LIN {X 0,Y 331.911,Z 733.66,A -85,B 0,C 180,E1 13527.132,E2 13527.132} C_VEL
LIN {X 0,Y 331.572,Z 733.66,A -85,B 0,C 180,E1 13534.718,E2 13534.718} C_VEL
LIN {X 0,Y 331.558,Z 733.66,A -85,B 0,C 180,E1 13538.128,E2 13538.128} C_VEL
LIN {X 0,Y 333.905,Z 739.259,A -85,B 0,C 180,E1 13538.848,E2 13538.848} C_VEL
LIN {X 0,Y 349.551,Z 763.487,A -85,B 0,C 180,E1 13542.624,E2 13542.624} C_VEL
LIN {X 0,Y 360.849,Z 785.15,A -85,B 0,C 180,E1 13545.118,E2 13545.118} C_VEL
LIN {X 0,Y 372.541,Z 822.08,A -85,B 0,C 180,E1 13548.359,E2 13548.359} C_VEL
LIN {X 0,Y 371.97,Z 832.356,A -85,B 0,C 180,E1 13548.893,E2 13548.893} C_VEL
LIN {X 0,Y 365.761,Z 868.683,A -85,B 0,C 180,E1 13551.046,E2 13551.046} C_VEL
LIN {X 0,Y 358.697,Z 901.168,A -85,B 0,C 180,E1 13553.962,E2 13553.962} C_VEL
LIN {X 0,Y 350.93,Z 932.25,A -85,B 0,C 180,E1 13557.955,E2 13557.955} C_VEL
LIN {X 0,Y 343.786,Z 958.969,A -85,B 0,C 180,E1 13562.81,E2 13562.81} C_VEL
LIN {X 0,Y 338.451,Z 980.705,A -85,B 0,C 180,E1 13568.341,E2 13568.341} C_VEL
LIN {X 0,Y 335.333,Z 997.025,A -85,B 0,C 180,E1 13574.281,E2 13574.281} C_VEL
LIN {X 0,Y 334.161,Z 1006.659,A -85,B 0,C 180,E1 13579.558,E2 13579.558} C_VEL
LIN {X 0,Y 333.965,Z 1012.316,A -85,B 0,C 180,E1 13584.797,E2 13584.797} C_VEL
LIN {X 0,Y 333.972,Z 1014.24,A -85,B 0,C 180,E1 13590,E2 13590} C_VEL
LIN {X 0,Y 333.994,Z 1012.324,A -85,B 0,C 180,E1 13595.202,E2 13595.202} C_VEL
LIN {X 0,Y 334.2,Z 1006.672,A -85,B 0,C 180,E1 13600.44,E2 13600.44} C_VEL
LIN {X 0,Y 335.673,Z 995.48,A -85,B 0,C 180,E1 13606.374,E2 13606.374} C_VEL
LIN {X 0,Y 339.032,Z 978.527,A -85,B 0,C 180,E1 13612.309,E2 13612.309} C_VEL
LIN {X 0,Y 344.609,Z 956.047,A -85,B 0,C 180,E1 13617.828,E2 13617.828} C_VEL
LIN {X 0,Y 345.475,Z 952.678,A -85,B 0,C 180,E1 13618.494,E2 13618.494} C_VEL
LIN {X 0,Y 344.782,Z 941.966,A -85,B 0,C 180,E1 13620.806,E2 13620.806} C_VEL
LIN {X 0,Y 344.477,Z 930.397,A -85,B 0,C 180,E1 13622.992,E2 13622.992} C_VEL
LIN {X 0,Y 352.645,Z 899.493,A -85,B 0,C 180,E1 13626.948,E2 13626.948} C_VEL
LIN {X 0,Y 360.081,Z 866.579,A -85,B 0,C 180,E1 13629.884,E2 13629.884} C_VEL
LIN {X 0,Y 366.33,Z 830.356,A -85,B 0,C 180,E1 13632.002,E2 13632.002} C_VEL
LIN {X 0,Y 366.745,Z 821.536,A -85,B 0,C 180,E1 13632.48,E2 13632.48} C_VEL
LIN {X 0,Y 363.263,Z 804.069,A -85,B 0,C 180,E1 13633.896,E2 13633.896} C_VEL
LIN {X 0,Y 362.721,Z 794.124,A -85,B 0,C 180,E1 13635.673,E2 13635.673} C_VEL
LIN {X 0,Y 360.552,Z 789.307,A -85,B 0,C 180,E1 13637.796,E2 13637.796} C_VEL
LIN {X 0,Y 359.041,Z 786.828,A -85,B 0,C 180,E1 13640.771,E2 13640.771} C_VEL
LIN {X 0,Y 359.521,Z 789.265,A -85,B 0,C 180,E1 13643.881,E2 13643.881} C_VEL
LIN {X 0,Y 360.829,Z 795.714,A -85,B 0,C 180,E1 13646.204,E2 13646.204} C_VEL
LIN {X 0,Y 361.355,Z 802.851,A -85,B 0,C 180,E1 13647.556,E2 13647.556} C_VEL
LIN {X 0,Y 354.669,Z 834.59,A -85,B 0,C 180,E1 13650.254,E2 13650.254} C_VEL
LIN {X 0,Y 348.457,Z 858.847,A -85,B 0,C 180,E1 13653.369,E2 13653.369} C_VEL
LIN {X 0,Y 342.32,Z 879.054,A -85,B 0,C 180,E1 13657.239,E2 13657.239} C_VEL
LIN {X 0,Y 336.926,Z 894.203,A -85,B 0,C 180,E1 13661.672,E2 13661.672} C_VEL
LIN {X 0,Y 332.546,Z 904.557,A -85,B 0,C 180,E1 13666.848,E2 13666.848} C_VEL
LIN {X 0,Y 329.992,Z 908.75,A -85,B 0,C 180,E1 13672.095,E2 13672.095} C_VEL
LIN {X 0,Y 328.809,Z 907.203,A -85,B 0,C 180,E1 13677.367,E2 13677.367} C_VEL
LIN {X 0,Y 328.812,Z 899.792,A -85,B 0,C 180,E1 13682.645,E2 13682.645} C_VEL
LIN {X 0,Y 329.842,Z 886.911,A -85,B 0,C 180,E1 13687.589,E2 13687.589} C_VEL
LIN {X 0,Y 331.846,Z 868.17,A -85,B 0,C 180,E1 13692.188,E2 13692.188} C_VEL
LIN {X 0,Y 334.313,Z 845.592,A -85,B 0,C 180,E1 13695.941,E2 13695.941} C_VEL
LIN {X 0,Y 337.167,Z 817.654,A -85,B 0,C 180,E1 13699.063,E2 13699.063} C_VEL
LIN {X 0,Y 339.255,Z 786.896,A -85,B 0,C 180,E1 13701.205,E2 13701.205} C_VEL
LIN {X 0,Y 324.043,Z 733.66,A -85,B 0,C 180,E1 13704.475,E2 13704.475} C_VEL
LIN {X 0,Y 323.746,Z 733.66,A -85,B 0,C 180,E1 13710.966,E2 13710.966} C_VEL
LIN {X 0,Y 323.642,Z 733.66,A -85,B 0,C 180,E1 13716.732,E2 13716.732} C_VEL
LIN {X 0,Y 325.686,Z 739.009,A -85,B 0,C 180,E1 13717.418,E2 13717.418} C_VEL
LIN {X 0,Y 329.033,Z 743.84,A -85,B 0,C 180,E1 13718.347,E2 13718.347} C_VEL
LIN {X 0,Y 345.773,Z 770.437,A -85,B 0,C 180,E1 13722.642,E2 13722.642} C_VEL
LIN {X 0,Y 358.943,Z 798.734,A -85,B 0,C 180,E1 13726.406,E2 13726.406} C_VEL
LIN {X 0,Y 365.577,Z 820.254,A -85,B 0,C 180,E1 13729.005,E2 13729.005} C_VEL
LIN {X 0,Y 359.079,Z 854.069,A -85,B 0,C 180,E1 13731.551,E2 13731.551} C_VEL
LIN {X 0,Y 351.407,Z 885.543,A -85,B 0,C 180,E1 13735.007,E2 13735.007} C_VEL
LIN {X 0,Y 343.459,Z 913.169,A -85,B 0,C 180,E1 13739.291,E2 13739.291} C_VEL
LIN {X 0,Y 336.444,Z 936.403,A -85,B 0,C 180,E1 13744.328,E2 13744.328} C_VEL
LIN {X 0,Y 330.909,Z 955.773,A -85,B 0,C 180,E1 13750.316,E2 13750.316} C_VEL
LIN {X 0,Y 327.668,Z 969.28,A -85,B 0,C 180,E1 13756.642,E2 13756.642} C_VEL
LIN {X 0,Y 326.169,Z 977.56,A -85,B 0,C 180,E1 13763.336,E2 13763.336} C_VEL
LIN {X 0,Y 325.999,Z 980.249,A -85,B 0,C 180,E1 13770,E2 13770} C_VEL
LIN {X 0,Y 326.191,Z 977.47,A -85,B 0,C 180,E1 13776.664,E2 13776.664} C_VEL
LIN {X 0,Y 327.718,Z 969.117,A -85,B 0,C 180,E1 13783.357,E2 13783.357} C_VEL
LIN {X 0,Y 331.009,Z 955.453,A -85,B 0,C 180,E1 13789.707,E2 13789.707} C_VEL
LIN {X 0,Y 336.625,Z 935.783,A -85,B 0,C 180,E1 13795.726,E2 13795.726} C_VEL
LIN {X 0,Y 343.667,Z 912.319,A -85,B 0,C 180,E1 13800.766,E2 13800.766} C_VEL
LIN {X 0,Y 351.73,Z 883.855,A -85,B 0,C 180,E1 13805.121,E2 13805.121} C_VEL
LIN {X 0,Y 359.385,Z 852.252,A -85,B 0,C 180,E1 13808.513,E2 13808.513} C_VEL
LIN {X 0,Y 365.542,Z 819.307,A -85,B 0,C 180,E1 13810.971,E2 13810.971} C_VEL
LIN {X 0,Y 355.171,Z 789.667,A -85,B 0,C 180,E1 13814.647,E2 13814.647} C_VEL
LIN {X 0,Y 340.019,Z 760.655,A -85,B 0,C 180,E1 13818.694,E2 13818.694} C_VEL
LIN {X 0,Y 326.225,Z 739.502,A -85,B 0,C 180,E1 13822.308,E2 13822.308} C_VEL
LIN {X 0,Y 323.762,Z 735.024,A -85,B 0,C 180,E1 13823.045,E2 13823.045} C_VEL
LIN {X 0,Y 323.659,Z 733.66,A -85,B 0,C 180,E1 13823.429,E2 13823.429} C_VEL
LIN {X 0,Y 323.752,Z 733.66,A -85,B 0,C 180,E1 13829.035,E2 13829.035} C_VEL
LIN {X 0,Y 324.019,Z 733.66,A -85,B 0,C 180,E1 13835.125,E2 13835.125} C_VEL
LIN {X 0,Y 324.332,Z 733.66,A -85,B 0,C 180,E1 13840.921,E2 13840.921} C_VEL
LIN {X 0,Y 324.702,Z 733.66,A -85,B 0,C 180,E1 13849.245,E2 13849.245} C_VEL
LIN {X 0,Y 325.441,Z 733.66,A -85,B 0,C 180,E1 13857.328,E2 13857.328} C_VEL
LIN {X 0,Y 325.436,Z 733.66,A -85,B 0,C 180,E1 13862.661,E2 13862.661} C_VEL
LIN {X 0,Y 324.793,Z 733.66,A -85,B 0,C 180,E1 13870.74,E2 13870.74} C_VEL
LIN {X 0,Y 324.346,Z 733.66,A -85,B 0,C 180,E1 13879.065,E2 13879.065} C_VEL
LIN {X 0,Y 323.972,Z 733.66,A -85,B 0,C 180,E1 13887.38,E2 13887.38} C_VEL
LIN {X 0,Y 323.64,Z 733.66,A -85,B 0,C 180,E1 13895.697,E2 13895.697} C_VEL
LIN {X 0,Y 323.716,Z 734.317,A -85,B 0,C 180,E1 13896.394,E2 13896.394} C_VEL
LIN {X 0,Y 326.473,Z 739.738,A -85,B 0,C 180,E1 13897.231,E2 13897.231} C_VEL
LIN {X 0,Y 343.183,Z 765.713,A -85,B 0,C 180,E1 13901.535,E2 13901.535} C_VEL
LIN {X 0,Y 355.345,Z 788.28,A -85,B 0,C 180,E1 13904.34,E2 13904.34} C_VEL
LIN {X 0,Y 366.252,Z 824.046,A -85,B 0,C 180,E1 13907.622,E2 13907.622} C_VEL
LIN {X 0,Y 366.021,Z 831.981,A -85,B 0,C 180,E1 13908.075,E2 13908.075} C_VEL
LIN {X 0,Y 359.568,Z 868.29,A -85,B 0,C 180,E1 13910.243,E2 13910.243} C_VEL
LIN {X 0,Y 352.248,Z 900.766,A -85,B 0,C 180,E1 13913.195,E2 13913.195} C_VEL
LIN {X 0,Y 344.17,Z 931.352,A -85,B 0,C 180,E1 13917.159,E2 13917.159} C_VEL
LIN {X 0,Y 336.58,Z 958.579,A -85,B 0,C 180,E1 13922.184,E2 13922.184} C_VEL
LIN {X 0,Y 330.923,Z 980.288,A -85,B 0,C 180,E1 13927.823,E2 13927.823} C_VEL
LIN {X 0,Y 327.586,Z 996.61,A -85,B 0,C 180,E1 13933.899,E2 13933.899} C_VEL
LIN {X 0,Y 326.289,Z 1006.247,A -85,B 0,C 180,E1 13939.303,E2 13939.303} C_VEL
LIN {X 0,Y 326.063,Z 1011.907,A -85,B 0,C 180,E1 13944.671,E2 13944.671} C_VEL
LIN {X 0,Y 326.088,Z 1013.834,A -85,B 0,C 180,E1 13950,E2 13950} C_VEL
LIN {X 0,Y 326.091,Z 1011.916,A -85,B 0,C 180,E1 13955.328,E2 13955.328} C_VEL
LIN {X 0,Y 326.331,Z 1006.261,A -85,B 0,C 180,E1 13960.695,E2 13960.695} C_VEL
LIN {X 0,Y 327.904,Z 995.065,A -85,B 0,C 180,E1 13966.773,E2 13966.773} C_VEL
LIN {X 0,Y 331.569,Z 978.115,A -85,B 0,C 180,E1 13972.839,E2 13972.839} C_VEL
LIN {X 0,Y 337.441,Z 955.636,A -85,B 0,C 180,E1 13978.472,E2 13978.472} C_VEL
LIN {X 0,Y 344.477,Z 930.397,A -85,B 0,C 180,E1 13982.992,E2 13982.992} C_VEL
LIN {X 0,Y 344.431,Z 918.196,A -85,B 0,C 180,E1 13985.076,E2 13985.076} C_VEL
LIN {X 0,Y 344.269,Z 907.016,A -85,B 0,C 180,E1 13986.843,E2 13986.843} C_VEL
LIN {X 0,Y 344.691,Z 905.27,A -85,B 0,C 180,E1 13987.058,E2 13987.058} C_VEL
LIN {X 0,Y 352.747,Z 871.938,A -85,B 0,C 180,E1 13990.276,E2 13990.276} C_VEL
LIN {X 0,Y 359.509,Z 835.875,A -85,B 0,C 180,E1 13992.57,E2 13992.57} C_VEL
LIN {X 0,Y 360.689,Z 824.185,A -85,B 0,C 180,E1 13993.179,E2 13993.179} C_VEL
LIN {X 0,Y 358.667,Z 809.134,A -85,B 0,C 180,E1 13994.518,E2 13994.518} C_VEL
LIN {X 0,Y 358.554,Z 799.927,A -85,B 0,C 180,E1 13996.276,E2 13996.276} C_VEL
LIN {X 0,Y 356.43,Z 795.267,A -85,B 0,C 180,E1 13998.867,E2 13998.867} C_VEL
LIN {X 0,Y 355.846,Z 794.198,A -85,B 0,C 180,E1 14000.349,E2 14000.349} C_VEL
LIN {X 0,Y 356.078,Z 796.729,A -85,B 0,C 180,E1 14003.891,E2 14003.891} C_VEL
LIN {X 0,Y 357.054,Z 804.029,A -85,B 0,C 180,E1 14006.282,E2 14006.282} C_VEL
LIN {X 0,Y 356.381,Z 808.267,A -85,B 0,C 180,E1 14006.789,E2 14006.789} C_VEL
LIN {X 0,Y 348.68,Z 839.669,A -85,B 0,C 180,E1 14009.69,E2 14009.69} C_VEL
LIN {X 0,Y 341.732,Z 863.695,A -85,B 0,C 180,E1 14013.037,E2 14013.037} C_VEL
LIN {X 0,Y 335.079,Z 883.09,A -85,B 0,C 180,E1 14017.07,E2 14017.07} C_VEL
LIN {X 0,Y 329.053,Z 898.034,A -85,B 0,C 180,E1 14021.912,E2 14021.912} C_VEL
LIN {X 0,Y 325.068,Z 906.383,A -85,B 0,C 180,E1 14026.54,E2 14026.54} C_VEL
LIN {X 0,Y 322.302,Z 910.263,A -85,B 0,C 180,E1 14031.905,E2 14031.905} C_VEL
LIN {X 0,Y 321.029,Z 908.48,A -85,B 0,C 180,E1 14037.303,E2 14037.303} C_VEL
LIN {X 0,Y 320.997,Z 900.823,A -85,B 0,C 180,E1 14042.709,E2 14042.709} C_VEL
LIN {X 0,Y 322.051,Z 887.692,A -85,B 0,C 180,E1 14047.774,E2 14047.774} C_VEL
LIN {X 0,Y 324.156,Z 868.679,A -85,B 0,C 180,E1 14052.481,E2 14052.481} C_VEL
LIN {X 0,Y 326.856,Z 844.616,A -85,B 0,C 180,E1 14056.488,E2 14056.488} C_VEL
LIN {X 0,Y 329.663,Z 817.872,A -85,B 0,C 180,E1 14059.477,E2 14059.477} C_VEL
LIN {X 0,Y 331.619,Z 787.21,A -85,B 0,C 180,E1 14061.647,E2 14061.647} C_VEL
LIN {X 0,Y 316.086,Z 733.66,A -85,B 0,C 180,E1 14065.038,E2 14065.038} C_VEL
LIN {X 0,Y 315.73,Z 733.66,A -85,B 0,C 180,E1 14073.573,E2 14073.573} C_VEL
